LIN {X 0,Y 371.44,Z 415.123,A -85,B 0,C 180,E1 -12712.236,E2 -12712.236} C_VEL
LIN {X 0,Y 371.913,Z 409.005,A -85,B 0,C 180,E1 -12713.675,E2 -12713.675} C_VEL
LIN {X 0,Y 370.1,Z 398.641,A -85,B 0,C 180,E1 -12716.295,E2 -12716.295} C_VEL
LIN {X 0,Y 369.046,Z 393.228,A -85,B 0,C 180,E1 -12717.735,E2 -12717.735} C_VEL
LIN {X 0,Y 368.911,Z 393.034,A -85,B 0,C 180,E1 -12720.987,E2 -12720.987} C_VEL
LIN {X 0,Y 368.937,Z 393.026,A -85,B 0,C 180,E1 -12724.853,E2 -12724.853} C_VEL
LIN {X 0,Y 368.91,Z 393.028,A -85,B 0,C 180,E1 -12728.64,E2 -12728.64} C_VEL
LIN {X 0,Y 368.881,Z 393.034,A -85,B 0,C 180,E1 -12732.009,E2 -12732.009} C_VEL
LIN {X 0,Y 368.953,Z 393.026,A -85,B 0,C 180,E1 -12735.187,E2 -12735.187} C_VEL
LIN {X 0,Y 368.939,Z 393.025,A -85,B 0,C 180,E1 -12738.185,E2 -12738.185} C_VEL
LIN {X 0,Y 368.912,Z 393.034,A -85,B 0,C 180,E1 -12741.358,E2 -12741.358} C_VEL
LIN {X 0,Y 368.934,Z 393.029,A -85,B 0,C 180,E1 -12745.146,E2 -12745.146} C_VEL
LIN {X 0,Y 368.926,Z 393.029,A -85,B 0,C 180,E1 -12749.046,E2 -12749.046} C_VEL
LIN {X 0,Y 368.976,Z 393.025,A -85,B 0,C 180,E1 -12751.563,E2 -12751.563} C_VEL
LIN {X 0,Y 368.996,Z 393.019,A -85,B 0,C 180,E1 -12754.019,E2 -12754.019} C_VEL
LIN {X 0,Y 368.92,Z 393.032,A -85,B 0,C 180,E1 -12757.604,E2 -12757.604} C_VEL
LIN {X 0,Y 368.978,Z 393.024,A -85,B 0,C 180,E1 -12761.107,E2 -12761.107} C_VEL
LIN {X 0,Y 368.993,Z 393.019,A -85,B 0,C 180,E1 -12764.535,E2 -12764.535} C_VEL
LIN {X 0,Y 368.999,Z 393.019,A -85,B 0,C 180,E1 -12767.906,E2 -12767.906} C_VEL
LIN {X 0,Y 369.161,Z 392.999,A -85,B 0,C 180,E1 -12771.869,E2 -12771.869} C_VEL
LIN {X 0,Y 369.138,Z 393.001,A -85,B 0,C 180,E1 -12774.537,E2 -12774.537} C_VEL
LIN {X 0,Y 369.313,Z 392.98,A -85,B 0,C 180,E1 -12777.819,E2 -12777.819} C_VEL
LIN {X 0,Y 369.453,Z 392.962,A -85,B 0,C 180,E1 -12780,E2 -12780} C_VEL
LIN {X 0,Y 369.314,Z 392.978,A -85,B 0,C 180,E1 -12782.181,E2 -12782.181} C_VEL
LIN {X 0,Y 369.192,Z 392.994,A -85,B 0,C 180,E1 -12786.614,E2 -12786.614} C_VEL
LIN {X 0,Y 369.062,Z 393.011,A -85,B 0,C 180,E1 -12789.868,E2 -12789.868} C_VEL
LIN {X 0,Y 369.032,Z 393.015,A -85,B 0,C 180,E1 -12793.772,E2 -12793.772} C_VEL
LIN {X 0,Y 368.996,Z 393.019,A -85,B 0,C 180,E1 -12797.769,E2 -12797.769} C_VEL
LIN {X 0,Y 368.924,Z 393.033,A -85,B 0,C 180,E1 -12801.22,E2 -12801.22} C_VEL
LIN {X 0,Y 368.953,Z 393.026,A -85,B 0,C 180,E1 -12804.776,E2 -12804.776} C_VEL
LIN {X 0,Y 368.983,Z 393.02,A -85,B 0,C 180,E1 -12808.436,E2 -12808.436} C_VEL
LIN {X 0,Y 368.896,Z 393.03,A -85,B 0,C 180,E1 -12812.238,E2 -12812.238} C_VEL
LIN {X 0,Y 368.926,Z 393.032,A -85,B 0,C 180,E1 -12815.002,E2 -12815.002} C_VEL
LIN {X 0,Y 368.907,Z 393.031,A -85,B 0,C 180,E1 -12818.641,E2 -12818.641} C_VEL
LIN {X 0,Y 368.879,Z 393.033,A -85,B 0,C 180,E1 -12822.01,E2 -12822.01} C_VEL
LIN {X 0,Y 368.905,Z 393.035,A -85,B 0,C 180,E1 -12825.18,E2 -12825.18} C_VEL
LIN {X 0,Y 368.908,Z 393.029,A -85,B 0,C 180,E1 -12828.182,E2 -12828.182} C_VEL
LIN {X 0,Y 368.912,Z 393.031,A -85,B 0,C 180,E1 -12831.359,E2 -12831.359} C_VEL
LIN {X 0,Y 368.936,Z 393.031,A -85,B 0,C 180,E1 -12835.147,E2 -12835.147} C_VEL
LIN {X 0,Y 368.929,Z 393.032,A -85,B 0,C 180,E1 -12839.047,E2 -12839.047} C_VEL
LIN {X 0,Y 368.976,Z 393.022,A -85,B 0,C 180,E1 -12841.564,E2 -12841.564} C_VEL
LIN {X 0,Y 369,Z 393.017,A -85,B 0,C 180,E1 -12844.02,E2 -12844.02} C_VEL
LIN {X 0,Y 368.933,Z 393.026,A -85,B 0,C 180,E1 -12847.605,E2 -12847.605} C_VEL
LIN {X 0,Y 368.959,Z 393.027,A -85,B 0,C 180,E1 -12851.106,E2 -12851.106} C_VEL
LIN {X 0,Y 368.999,Z 393.02,A -85,B 0,C 180,E1 -12854.535,E2 -12854.535} C_VEL
LIN {X 0,Y 369.086,Z 393.119,A -85,B 0,C 180,E1 -12857.281,E2 -12857.281} C_VEL
LIN {X 0,Y 371.157,Z 404.31,A -85,B 0,C 180,E1 -12860.381,E2 -12860.381} C_VEL
LIN {X 0,Y 371.305,Z 407.805,A -85,B 0,C 180,E1 -12861.291,E2 -12861.291} C_VEL
LIN {X 0,Y 370.959,Z 411.278,A -85,B 0,C 180,E1 -12862.105,E2 -12862.105} C_VEL
LIN {X 0,Y 371.664,Z 415.551,A -85,B 0,C 180,E1 -12862.281,E2 -12862.281} C_VEL
LIN {X 0,Y 375.657,Z 437.442,A -85,B 0,C 180,E1 -12862.901,E2 -12862.901} C_VEL
LIN {X 0,Y 374.451,Z 518.084,A -85,B 0,C 180,E1 -12864.459,E2 -12864.459} C_VEL
LIN {X 0,Y 373.984,Z 531.756,A -85,B 0,C 180,E1 -12864.943,E2 -12864.943} C_VEL
LIN {X 0,Y 373.319,Z 544.448,A -85,B 0,C 180,E1 -12865.614,E2 -12865.614} C_VEL
LIN {X 0,Y 372.489,Z 556.486,A -85,B 0,C 180,E1 -12866.484,E2 -12866.484} C_VEL
LIN {X 0,Y 371.473,Z 567.981,A -85,B 0,C 180,E1 -12867.56,E2 -12867.56} C_VEL
LIN {X 0,Y 370.657,Z 578.297,A -85,B 0,C 180,E1 -12868.777,E2 -12868.777} C_VEL
LIN {X 0,Y 369.86,Z 586.759,A -85,B 0,C 180,E1 -12870,E2 -12870} C_VEL
LIN {X 0,Y 368.966,Z 595.93,A -85,B 0,C 180,E1 -12871.637,E2 -12871.637} C_VEL
LIN {X 0,Y 368.405,Z 603.301,A -85,B 0,C 180,E1 -12873.281,E2 -12873.281} C_VEL
LIN {X 0,Y 367.91,Z 609.23,A -85,B 0,C 180,E1 -12874.931,E2 -12874.931} C_VEL
LIN {X 0,Y 367.727,Z 613.898,A -85,B 0,C 180,E1 -12876.584,E2 -12876.584} C_VEL
LIN {X 0,Y 367.471,Z 617.474,A -85,B 0,C 180,E1 -12878.246,E2 -12878.246} C_VEL
LIN {X 0,Y 367.268,Z 620.03,A -85,B 0,C 180,E1 -12879.917,E2 -12879.917} C_VEL
LIN {X 0,Y 367.283,Z 621.209,A -85,B 0,C 180,E1 -12881.031,E2 -12881.031} C_VEL
LIN {X 0,Y 367.292,Z 622.145,A -85,B 0,C 180,E1 -12882.613,E2 -12882.613} C_VEL
LIN {X 0,Y 367.18,Z 622.222,A -85,B 0,C 180,E1 -12884.407,E2 -12884.407} C_VEL
LIN {X 0,Y 367.228,Z 621.72,A -85,B 0,C 180,E1 -12885.541,E2 -12885.541} C_VEL
LIN {X 0,Y 367.353,Z 620.477,A -85,B 0,C 180,E1 -12886.973,E2 -12886.973} C_VEL
LIN {X 0,Y 367.665,Z 617.626,A -85,B 0,C 180,E1 -12888.962,E2 -12888.962} C_VEL
LIN {X 0,Y 368.017,Z 614.077,A -85,B 0,C 180,E1 -12890.65,E2 -12890.65} C_VEL
LIN {X 0,Y 368.293,Z 611.729,A -85,B 0,C 180,E1 -12891.537,E2 -12891.537} C_VEL
LIN {X 0,Y 367.938,Z 609.343,A -85,B 0,C 180,E1 -12892.375,E2 -12892.375} C_VEL
LIN {X 0,Y 365.697,Z 605.131,A -85,B 0,C 180,E1 -12893.734,E2 -12893.734} C_VEL
LIN {X 0,Y 363.513,Z 600.325,A -85,B 0,C 180,E1 -12895.054,E2 -12895.054} C_VEL
LIN {X 0,Y 363.247,Z 596.96,A -85,B 0,C 180,E1 -12895.819,E2 -12895.819} C_VEL
LIN {X 0,Y 364.426,Z 588.08,A -85,B 0,C 180,E1 -12897.487,E2 -12897.487} C_VEL
LIN {X 0,Y 365.716,Z 577.768,A -85,B 0,C 180,E1 -12899.027,E2 -12899.027} C_VEL
LIN {X 0,Y 367.063,Z 567.317,A -85,B 0,C 180,E1 -12900.261,E2 -12900.261} C_VEL
LIN {X 0,Y 368.253,Z 555.954,A -85,B 0,C 180,E1 -12901.335,E2 -12901.335} C_VEL
LIN {X 0,Y 369.319,Z 544.043,A -85,B 0,C 180,E1 -12902.196,E2 -12902.196} C_VEL
LIN {X 0,Y 370.206,Z 531.197,A -85,B 0,C 180,E1 -12902.875,E2 -12902.875} C_VEL
LIN {X 0,Y 370.844,Z 517.98,A -85,B 0,C 180,E1 -12903.338,E2 -12903.338} C_VEL
LIN {X 0,Y 372.433,Z 439.897,A -85,B 0,C 180,E1 -12904.888,E2 -12904.888} C_VEL
LIN {X 0,Y 367.754,Z 418.56,A -85,B 0,C 180,E1 -12905.694,E2 -12905.694} C_VEL
LIN {X 0,Y 365.867,Z 412.519,A -85,B 0,C 180,E1 -12905.985,E2 -12905.985} C_VEL
LIN {X 0,Y 365.515,Z 411.249,A -85,B 0,C 180,E1 -12906.142,E2 -12906.142} C_VEL
LIN {X 0,Y 363.427,Z 400.528,A -85,B 0,C 180,E1 -12909.328,E2 -12909.328} C_VEL
LIN {X 0,Y 361.906,Z 393.937,A -85,B 0,C 180,E1 -12911.48,E2 -12911.48} C_VEL
LIN {X 0,Y 361.929,Z 393.903,A -85,B 0,C 180,E1 -12914.35,E2 -12914.35} C_VEL
LIN {X 0,Y 361.882,Z 393.901,A -85,B 0,C 180,E1 -12917.559,E2 -12917.559} C_VEL
LIN {X 0,Y 361.869,Z 393.901,A -85,B 0,C 180,E1 -12920.972,E2 -12920.972} C_VEL
LIN {X 0,Y 361.869,Z 393.9,A -85,B 0,C 180,E1 -12924.654,E2 -12924.654} C_VEL
LIN {X 0,Y 361.853,Z 393.911,A -85,B 0,C 180,E1 -12928.372,E2 -12928.372} C_VEL
LIN {X 0,Y 361.915,Z 393.9,A -85,B 0,C 180,E1 -12932.222,E2 -12932.222} C_VEL
LIN {X 0,Y 361.921,Z 393.9,A -85,B 0,C 180,E1 -12934.709,E2 -12934.709} C_VEL
LIN {X 0,Y 361.894,Z 393.899,A -85,B 0,C 180,E1 -12938.347,E2 -12938.347} C_VEL
LIN {X 0,Y 361.96,Z 393.891,A -85,B 0,C 180,E1 -12942.061,E2 -12942.061} C_VEL
LIN {X 0,Y 361.99,Z 393.886,A -85,B 0,C 180,E1 -12946.101,E2 -12946.101} C_VEL
LIN {X 0,Y 362.028,Z 393.879,A -85,B 0,C 180,E1 -12949.938,E2 -12949.938} C_VEL
LIN {X 0,Y 362.143,Z 393.874,A -85,B 0,C 180,E1 -12952.192,E2 -12952.192} C_VEL
LIN {X 0,Y 362.111,Z 393.87,A -85,B 0,C 180,E1 -12954.431,E2 -12954.431} C_VEL
LIN {X 0,Y 362.282,Z 393.853,A -85,B 0,C 180,E1 -12957.777,E2 -12957.777} C_VEL
LIN {X 0,Y 362.421,Z 393.833,A -85,B 0,C 180,E1 -12960,E2 -12960} C_VEL
LIN {X 0,Y 362.275,Z 393.857,A -85,B 0,C 180,E1 -12962.224,E2 -12962.224} C_VEL
LIN {X 0,Y 362.164,Z 393.875,A -85,B 0,C 180,E1 -12966.686,E2 -12966.686} C_VEL
LIN {X 0,Y 362.067,Z 393.877,A -85,B 0,C 180,E1 -12968.934,E2 -12968.934} C_VEL
LIN {X 0,Y 361.959,Z 393.898,A -85,B 0,C 180,E1 -12972.332,E2 -12972.332} C_VEL
LIN {X 0,Y 361.954,Z 393.892,A -85,B 0,C 180,E1 -12974.621,E2 -12974.621} C_VEL
LIN {X 0,Y 361.952,Z 393.891,A -85,B 0,C 180,E1 -12978.1,E2 -12978.1} C_VEL
LIN {X 0,Y 361.885,Z 393.902,A -85,B 0,C 180,E1 -12981.653,E2 -12981.653} C_VEL
LIN {X 0,Y 361.921,Z 393.9,A -85,B 0,C 180,E1 -12985.291,E2 -12985.291} C_VEL
LIN {X 0,Y 361.912,Z 393.899,A -85,B 0,C 180,E1 -12987.779,E2 -12987.779} C_VEL
LIN {X 0,Y 361.841,Z 393.91,A -85,B 0,C 180,E1 -12991.286,E2 -12991.286} C_VEL
LIN {X 0,Y 361.849,Z 393.907,A -85,B 0,C 180,E1 -12994.281,E2 -12994.281} C_VEL
LIN {X 0,Y 361.861,Z 393.905,A -85,B 0,C 180,E1 -12997.224,E2 -12997.224} C_VEL
LIN {X 0,Y 361.901,Z 393.89,A -85,B 0,C 180,E1 -13000.769,E2 -13000.769} C_VEL
LIN {X 0,Y 361.907,Z 393.907,A -85,B 0,C 180,E1 -13004.355,E2 -13004.355} C_VEL
LIN {X 0,Y 361.837,Z 393.91,A -85,B 0,C 180,E1 -13007.568,E2 -13007.568} C_VEL
LIN {X 0,Y 361.869,Z 393.905,A -85,B 0,C 180,E1 -13010.974,E2 -13010.974} C_VEL
LIN {X 0,Y 361.873,Z 393.91,A -85,B 0,C 180,E1 -13014.656,E2 -13014.656} C_VEL
LIN {X 0,Y 361.836,Z 393.91,A -85,B 0,C 180,E1 -13018.371,E2 -13018.371} C_VEL
LIN {X 0,Y 361.93,Z 394.09,A -85,B 0,C 180,E1 -13019.602,E2 -13019.602} C_VEL
LIN {X 0,Y 364.258,Z 403.929,A -85,B 0,C 180,E1 -13022.564,E2 -13022.564} C_VEL
LIN {X 0,Y 366.125,Z 413.741,A -85,B 0,C 180,E1 -13025.324,E2 -13025.324} C_VEL
LIN {X 0,Y 366.107,Z 417.243,A -85,B 0,C 180,E1 -13026.227,E2 -13026.227} C_VEL
LIN {X 0,Y 365.803,Z 420.538,A -85,B 0,C 180,E1 -13026.993,E2 -13026.993} C_VEL
LIN {X 0,Y 366.882,Z 425.74,A -85,B 0,C 180,E1 -13027.244,E2 -13027.244} C_VEL
LIN {X 0,Y 370.779,Z 444.027,A -85,B 0,C 180,E1 -13027.928,E2 -13027.928} C_VEL
LIN {X 0,Y 372.23,Z 453.66,A -85,B 0,C 180,E1 -13028.238,E2 -13028.238} C_VEL
LIN {X 0,Y 370.734,Z 528.187,A -85,B 0,C 180,E1 -13029.724,E2 -13029.724} C_VEL
LIN {X 0,Y 370.096,Z 541.357,A -85,B 0,C 180,E1 -13030.194,E2 -13030.194} C_VEL
LIN {X 0,Y 369.108,Z 553.473,A -85,B 0,C 180,E1 -13030.826,E2 -13030.826} C_VEL
LIN {X 0,Y 368.082,Z 564.883,A -85,B 0,C 180,E1 -13031.637,E2 -13031.637} C_VEL
LIN {X 0,Y 366.916,Z 575.332,A -85,B 0,C 180,E1 -13032.586,E2 -13032.586} C_VEL
LIN {X 0,Y 365.592,Z 586.073,A -85,B 0,C 180,E1 -13033.816,E2 -13033.816} C_VEL
LIN {X 0,Y 364.426,Z 595.862,A -85,B 0,C 180,E1 -13035.217,E2 -13035.217} C_VEL
LIN {X 0,Y 363.392,Z 603.678,A -85,B 0,C 180,E1 -13036.581,E2 -13036.581} C_VEL
LIN {X 0,Y 362.314,Z 611.495,A -85,B 0,C 180,E1 -13038.249,E2 -13038.249} C_VEL
LIN {X 0,Y 361.558,Z 617.752,A -85,B 0,C 180,E1 -13039.925,E2 -13039.925} C_VEL
LIN {X 0,Y 360.939,Z 622.747,A -85,B 0,C 180,E1 -13041.603,E2 -13041.603} C_VEL
LIN {X 0,Y 360.582,Z 626.625,A -85,B 0,C 180,E1 -13043.285,E2 -13043.285} C_VEL
LIN {X 0,Y 360.381,Z 630.221,A -85,B 0,C 180,E1 -13045.526,E2 -13045.526} C_VEL
LIN {X 0,Y 360.279,Z 631.412,A -85,B 0,C 180,E1 -13046.645,E2 -13046.645} C_VEL
LIN {X 0,Y 360.249,Z 632.531,A -85,B 0,C 180,E1 -13048.882,E2 -13048.882} C_VEL
LIN {X 0,Y 360.29,Z 632.513,A -85,B 0,C 180,E1 -13050,E2 -13050} C_VEL
LIN {X 0,Y 360.251,Z 632.109,A -85,B 0,C 180,E1 -13051.118,E2 -13051.118} C_VEL
LIN {X 0,Y 360.226,Z 631.272,A -85,B 0,C 180,E1 -13052.236,E2 -13052.236} C_VEL
LIN {X 0,Y 360.275,Z 630.026,A -85,B 0,C 180,E1 -13053.355,E2 -13053.355} C_VEL
LIN {X 0,Y 360.353,Z 627.374,A -85,B 0,C 180,E1 -13055.035,E2 -13055.035} C_VEL
LIN {X 0,Y 360.501,Z 623.694,A -85,B 0,C 180,E1 -13056.717,E2 -13056.717} C_VEL
LIN {X 0,Y 360.837,Z 618.886,A -85,B 0,C 180,E1 -13058.4,E2 -13058.4} C_VEL
LIN {X 0,Y 361.294,Z 612.8,A -85,B 0,C 180,E1 -13060.083,E2 -13060.083} C_VEL
LIN {X 0,Y 361.948,Z 605.214,A -85,B 0,C 180,E1 -13061.764,E2 -13061.764} C_VEL
LIN {X 0,Y 362.734,Z 597.46,A -85,B 0,C 180,E1 -13063.159,E2 -13063.159} C_VEL
LIN {X 0,Y 363.644,Z 587.98,A -85,B 0,C 180,E1 -13064.551,E2 -13064.551} C_VEL
LIN {X 0,Y 364.507,Z 577.427,A -85,B 0,C 180,E1 -13065.804,E2 -13065.804} C_VEL
LIN {X 0,Y 365.426,Z 565.676,A -85,B 0,C 180,E1 -13066.911,E2 -13066.911} C_VEL
LIN {X 0,Y 366.366,Z 553.12,A -85,B 0,C 180,E1 -13067.802,E2 -13067.802} C_VEL
LIN {X 0,Y 367.121,Z 539.852,A -85,B 0,C 180,E1 -13068.485,E2 -13068.485} C_VEL
LIN {X 0,Y 367.589,Z 527.842,A -85,B 0,C 180,E1 -13068.895,E2 -13068.895} C_VEL
LIN {X 0,Y 368.647,Z 450.626,A -85,B 0,C 180,E1 -13070.418,E2 -13070.418} C_VEL
LIN {X 0,Y 364.072,Z 420.84,A -85,B 0,C 180,E1 -13071.276,E2 -13071.276} C_VEL
LIN {X 0,Y 364.923,Z 411.05,A -85,B 0,C 180,E1 -13073.554,E2 -13073.554} C_VEL
LIN {X 0,Y 364.068,Z 404.839,A -85,B 0,C 180,E1 -13075.131,E2 -13075.131} C_VEL
LIN {X 0,Y 362.017,Z 394.269,A -85,B 0,C 180,E1 -13077.927,E2 -13077.927} C_VEL
LIN {X 0,Y 361.946,Z 393.899,A -85,B 0,C 180,E1 -13078.248,E2 -13078.248} C_VEL
LIN {X 0,Y 361.838,Z 393.915,A -85,B 0,C 180,E1 -13081.629,E2 -13081.629} C_VEL
LIN {X 0,Y 361.875,Z 393.909,A -85,B 0,C 180,E1 -13085.344,E2 -13085.344} C_VEL
LIN {X 0,Y 361.871,Z 393.907,A -85,B 0,C 180,E1 -13089.026,E2 -13089.026} C_VEL
LIN {X 0,Y 361.838,Z 393.91,A -85,B 0,C 180,E1 -13092.828,E2 -13092.828} C_VEL
LIN {X 0,Y 361.897,Z 393.904,A -85,B 0,C 180,E1 -13095.933,E2 -13095.933} C_VEL
LIN {X 0,Y 361.903,Z 393.905,A -85,B 0,C 180,E1 -13099.231,E2 -13099.231} C_VEL
LIN {X 0,Y 361.867,Z 393.908,A -85,B 0,C 180,E1 -13102.982,E2 -13102.982} C_VEL
LIN {X 0,Y 361.856,Z 393.907,A -85,B 0,C 180,E1 -13106.63,E2 -13106.63} C_VEL
LIN {X 0,Y 361.871,Z 393.909,A -85,B 0,C 180,E1 -13109.672,E2 -13109.672} C_VEL
LIN {X 0,Y 361.951,Z 393.901,A -85,B 0,C 180,E1 -13113.475,E2 -13113.475} C_VEL
LIN {X 0,Y 361.878,Z 393.908,A -85,B 0,C 180,E1 -13117.144,E2 -13117.144} C_VEL
LIN {X 0,Y 361.916,Z 393.9,A -85,B 0,C 180,E1 -13120.724,E2 -13120.724} C_VEL
LIN {X 0,Y 361.941,Z 393.897,A -85,B 0,C 180,E1 -13124.226,E2 -13124.226} C_VEL
LIN {X 0,Y 361.994,Z 393.89,A -85,B 0,C 180,E1 -13126.528,E2 -13126.528} C_VEL
LIN {X 0,Y 362.026,Z 393.887,A -85,B 0,C 180,E1 -13129.938,E2 -13129.938} C_VEL
LIN {X 0,Y 362.157,Z 393.876,A -85,B 0,C 180,E1 -13133.313,E2 -13133.313} C_VEL
LIN {X 0,Y 362.277,Z 393.857,A -85,B 0,C 180,E1 -13137.776,E2 -13137.776} C_VEL
LIN {X 0,Y 362.422,Z 393.837,A -85,B 0,C 180,E1 -13140,E2 -13140} C_VEL
LIN {X 0,Y 362.278,Z 393.855,A -85,B 0,C 180,E1 -13142.223,E2 -13142.223} C_VEL
LIN {X 0,Y 362.159,Z 393.871,A -85,B 0,C 180,E1 -13146.686,E2 -13146.686} C_VEL
LIN {X 0,Y 362.026,Z 393.886,A -85,B 0,C 180,E1 -13150.062,E2 -13150.062} C_VEL
LIN {X 0,Y 361.993,Z 393.891,A -85,B 0,C 180,E1 -13153.899,E2 -13153.899} C_VEL
LIN {X 0,Y 361.963,Z 393.894,A -85,B 0,C 180,E1 -13157.939,E2 -13157.939} C_VEL
LIN {X 0,Y 361.887,Z 393.905,A -85,B 0,C 180,E1 -13161.653,E2 -13161.653} C_VEL
LIN {X 0,Y 361.924,Z 393.904,A -85,B 0,C 180,E1 -13165.29,E2 -13165.29} C_VEL
LIN {X 0,Y 361.919,Z 393.9,A -85,B 0,C 180,E1 -13167.778,E2 -13167.778} C_VEL
LIN {X 0,Y 361.843,Z 393.914,A -85,B 0,C 180,E1 -13171.286,E2 -13171.286} C_VEL
LIN {X 0,Y 361.851,Z 393.908,A -85,B 0,C 180,E1 -13174.281,E2 -13174.281} C_VEL
LIN {X 0,Y 361.862,Z 393.912,A -85,B 0,C 180,E1 -13177.224,E2 -13177.224} C_VEL
LIN {X 0,Y 361.833,Z 393.913,A -85,B 0,C 180,E1 -13180.756,E2 -13180.756} C_VEL
LIN {X 0,Y 361.832,Z 393.911,A -85,B 0,C 180,E1 -13184.366,E2 -13184.366} C_VEL
LIN {X 0,Y 361.854,Z 393.909,A -85,B 0,C 180,E1 -13187.565,E2 -13187.565} C_VEL
LIN {X 0,Y 361.874,Z 393.911,A -85,B 0,C 180,E1 -13190.973,E2 -13190.973} C_VEL
LIN {X 0,Y 361.874,Z 393.908,A -85,B 0,C 180,E1 -13194.655,E2 -13194.655} C_VEL
LIN {X 0,Y 361.837,Z 393.91,A -85,B 0,C 180,E1 -13198.371,E2 -13198.371} C_VEL
LIN {X 0,Y 361.9,Z 393.908,A -85,B 0,C 180,E1 -13200.956,E2 -13200.956} C_VEL
LIN {X 0,Y 361.954,Z 393.897,A -85,B 0,C 180,E1 -13203.475,E2 -13203.475} C_VEL
LIN {X 0,Y 361.891,Z 393.907,A -85,B 0,C 180,E1 -13207.145,E2 -13207.145} C_VEL
LIN {X 0,Y 361.908,Z 393.905,A -85,B 0,C 180,E1 -13210.724,E2 -13210.724} C_VEL
LIN {X 0,Y 361.934,Z 393.902,A -85,B 0,C 180,E1 -13213.066,E2 -13213.066} C_VEL
LIN {X 0,Y 362.053,Z 393.976,A -85,B 0,C 180,E1 -13217.03,E2 -13217.03} C_VEL
LIN {X 0,Y 364.341,Z 406.519,A -85,B 0,C 180,E1 -13220.563,E2 -13220.563} C_VEL
LIN {X 0,Y 364.143,Z 411.267,A -85,B 0,C 180,E1 -13221.747,E2 -13221.747} C_VEL
LIN {X 0,Y 364.313,Z 413.493,A -85,B 0,C 180,E1 -13221.875,E2 -13221.875} C_VEL
LIN {X 0,Y 368.927,Z 439.229,A -85,B 0,C 180,E1 -13222.618,E2 -13222.618} C_VEL
LIN {X 0,Y 367.614,Z 518.872,A -85,B 0,C 180,E1 -13224.188,E2 -13224.188} C_VEL
LIN {X 0,Y 367.077,Z 532.529,A -85,B 0,C 180,E1 -13224.689,E2 -13224.689} C_VEL
LIN {X 0,Y 366.387,Z 545.345,A -85,B 0,C 180,E1 -13225.392,E2 -13225.392} C_VEL
LIN {X 0,Y 365.544,Z 557.165,A -85,B 0,C 180,E1 -13226.279,E2 -13226.279} C_VEL
LIN {X 0,Y 364.495,Z 568.557,A -85,B 0,C 180,E1 -13227.375,E2 -13227.375} C_VEL
LIN {X 0,Y 363.656,Z 578.783,A -85,B 0,C 180,E1 -13228.615,E2 -13228.615} C_VEL
LIN {X 0,Y 362.751,Z 587.996,A -85,B 0,C 180,E1 -13230,E2 -13230} C_VEL
LIN {X 0,Y 361.864,Z 596.958,A -85,B 0,C 180,E1 -13231.669,E2 -13231.669} C_VEL
LIN {X 0,Y 361.29,Z 604.167,A -85,B 0,C 180,E1 -13233.345,E2 -13233.345} C_VEL
LIN {X 0,Y 360.824,Z 609.932,A -85,B 0,C 180,E1 -13235.028,E2 -13235.028} C_VEL
LIN {X 0,Y 360.596,Z 614.466,A -85,B 0,C 180,E1 -13236.715,E2 -13236.715} C_VEL
LIN {X 0,Y 360.438,Z 616.864,A -85,B 0,C 180,E1 -13237.844,E2 -13237.844} C_VEL
LIN {X 0,Y 360.268,Z 618.833,A -85,B 0,C 180,E1 -13238.978,E2 -13238.978} C_VEL
LIN {X 0,Y 360.163,Z 620.376,A -85,B 0,C 180,E1 -13240.114,E2 -13240.114} C_VEL
LIN {X 0,Y 360.177,Z 621.451,A -85,B 0,C 180,E1 -13241.252,E2 -13241.252} C_VEL
LIN {X 0,Y 360.205,Z 622.257,A -85,B 0,C 180,E1 -13242.695,E2 -13242.695} C_VEL
LIN {X 0,Y 360.095,Z 622.269,A -85,B 0,C 180,E1 -13244.697,E2 -13244.697} C_VEL
LIN {X 0,Y 360.167,Z 621.68,A -85,B 0,C 180,E1 -13245.853,E2 -13245.853} C_VEL
LIN {X 0,Y 360.297,Z 620.6,A -85,B 0,C 180,E1 -13247.098,E2 -13247.098} C_VEL
LIN {X 0,Y 360.45,Z 619.268,A -85,B 0,C 180,E1 -13248.177,E2 -13248.177} C_VEL
LIN {X 0,Y 360.768,Z 616.239,A -85,B 0,C 180,E1 -13249.932,E2 -13249.932} C_VEL
LIN {X 0,Y 361.261,Z 612.074,A -85,B 0,C 180,E1 -13251.692,E2 -13251.692} C_VEL
LIN {X 0,Y 362.046,Z 605.568,A -85,B 0,C 180,E1 -13253.752,E2 -13253.752} C_VEL
LIN {X 0,Y 363.006,Z 598.411,A -85,B 0,C 180,E1 -13255.516,E2 -13255.516} C_VEL
LIN {X 0,Y 363.247,Z 596.96,A -85,B 0,C 180,E1 -13255.819,E2 -13255.819} C_VEL
LIN {X 0,Y 362.999,Z 593.432,A -85,B 0,C 180,E1 -13256.567,E2 -13256.567} C_VEL
LIN {X 0,Y 360.979,Z 587.458,A -85,B 0,C 180,E1 -13257.786,E2 -13257.786} C_VEL
LIN {X 0,Y 359.151,Z 580.987,A -85,B 0,C 180,E1 -13258.94,E2 -13258.94} C_VEL
LIN {X 0,Y 359.183,Z 576.611,A -85,B 0,C 180,E1 -13259.572,E2 -13259.572} C_VEL
LIN {X 0,Y 360.606,Z 565.776,A -85,B 0,C 180,E1 -13260.84,E2 -13260.84} C_VEL
LIN {X 0,Y 361.725,Z 555.469,A -85,B 0,C 180,E1 -13261.803,E2 -13261.803} C_VEL
LIN {X 0,Y 362.819,Z 543.335,A -85,B 0,C 180,E1 -13262.679,E2 -13262.679} C_VEL
LIN {X 0,Y 363.766,Z 530.221,A -85,B 0,C 180,E1 -13263.367,E2 -13263.367} C_VEL
LIN {X 0,Y 364.398,Z 517.585,A -85,B 0,C 180,E1 -13263.799,E2 -13263.799} C_VEL
LIN {X 0,Y 365.977,Z 440.622,A -85,B 0,C 180,E1 -13265.354,E2 -13265.354} C_VEL
LIN {X 0,Y 361.106,Z 418.719,A -85,B 0,C 180,E1 -13266.218,E2 -13266.218} C_VEL
LIN {X 0,Y 358.451,Z 411.884,A -85,B 0,C 180,E1 -13266.627,E2 -13266.627} C_VEL
LIN {X 0,Y 357.191,Z 405.438,A -85,B 0,C 180,E1 -13268.506,E2 -13268.506} C_VEL
LIN {X 0,Y 355.277,Z 396.751,A -85,B 0,C 180,E1 -13271.262,E2 -13271.262} C_VEL
LIN {X 0,Y 354.868,Z 394.807,A -85,B 0,C 180,E1 -13271.983,E2 -13271.983} C_VEL
LIN {X 0,Y 354.883,Z 394.775,A -85,B 0,C 180,E1 -13275.473,E2 -13275.473} C_VEL
LIN {X 0,Y 354.851,Z 394.783,A -85,B 0,C 180,E1 -13279.188,E2 -13279.188} C_VEL
LIN {X 0,Y 354.804,Z 394.786,A -85,B 0,C 180,E1 -13282.401,E2 -13282.401} C_VEL
LIN {X 0,Y 354.806,Z 394.777,A -85,B 0,C 180,E1 -13284.94,E2 -13284.94} C_VEL
LIN {X 0,Y 354.809,Z 394.789,A -85,B 0,C 180,E1 -13288.399,E2 -13288.399} C_VEL
LIN {X 0,Y 354.847,Z 394.777,A -85,B 0,C 180,E1 -13291.619,E2 -13291.619} C_VEL
LIN {X 0,Y 354.892,Z 394.776,A -85,B 0,C 180,E1 -13294.172,E2 -13294.172} C_VEL
LIN {X 0,Y 354.834,Z 394.778,A -85,B 0,C 180,E1 -13297.894,E2 -13297.894} C_VEL
LIN {X 0,Y 354.916,Z 394.768,A -85,B 0,C 180,E1 -13301.891,E2 -13301.891} C_VEL
LIN {X 0,Y 354.935,Z 394.765,A -85,B 0,C 180,E1 -13305.981,E2 -13305.981} C_VEL
LIN {X 0,Y 354.975,Z 394.757,A -85,B 0,C 180,E1 -13309.736,E2 -13309.736} C_VEL
LIN {X 0,Y 355.106,Z 394.75,A -85,B 0,C 180,E1 -13312.037,E2 -13312.037} C_VEL
LIN {X 0,Y 355.086,Z 394.745,A -85,B 0,C 180,E1 -13314.321,E2 -13314.321} C_VEL
LIN {X 0,Y 355.246,Z 394.73,A -85,B 0,C 180,E1 -13317.732,E2 -13317.732} C_VEL
LIN {X 0,Y 355.391,Z 394.709,A -85,B 0,C 180,E1 -13320,E2 -13320} C_VEL
LIN {X 0,Y 355.238,Z 394.734,A -85,B 0,C 180,E1 -13322.268,E2 -13322.268} C_VEL
LIN {X 0,Y 355.13,Z 394.749,A -85,B 0,C 180,E1 -13326.819,E2 -13326.819} C_VEL
LIN {X 0,Y 355.009,Z 394.756,A -85,B 0,C 180,E1 -13329.113,E2 -13329.113} C_VEL
LIN {X 0,Y 354.919,Z 394.771,A -85,B 0,C 180,E1 -13332.581,E2 -13332.581} C_VEL
LIN {X 0,Y 354.882,Z 394.778,A -85,B 0,C 180,E1 -13336.096,E2 -13336.096} C_VEL
LIN {X 0,Y 354.899,Z 394.769,A -85,B 0,C 180,E1 -13338.472,E2 -13338.472} C_VEL
LIN {X 0,Y 354.828,Z 394.782,A -85,B 0,C 180,E1 -13342.107,E2 -13342.107} C_VEL
LIN {X 0,Y 354.892,Z 394.775,A -85,B 0,C 180,E1 -13345.828,E2 -13345.828} C_VEL
LIN {X 0,Y 354.848,Z 394.78,A -85,B 0,C 180,E1 -13349.679,E2 -13349.679} C_VEL
LIN {X 0,Y 354.801,Z 394.785,A -85,B 0,C 180,E1 -13353.703,E2 -13353.703} C_VEL
LIN {X 0,Y 354.794,Z 394.79,A -85,B 0,C 180,E1 -13356.46,E2 -13356.46} C_VEL
LIN {X 0,Y 354.819,Z 394.785,A -85,B 0,C 180,E1 -13359.425,E2 -13359.425} C_VEL
LIN {X 0,Y 354.831,Z 394.777,A -85,B 0,C 180,E1 -13362.876,E2 -13362.876} C_VEL
LIN {X 0,Y 354.78,Z 394.78,A -85,B 0,C 180,E1 -13366.107,E2 -13366.107} C_VEL
LIN {X 0,Y 354.804,Z 394.785,A -85,B 0,C 180,E1 -13369.183,E2 -13369.183} C_VEL
LIN {X 0,Y 354.806,Z 394.788,A -85,B 0,C 180,E1 -13372.403,E2 -13372.403} C_VEL
LIN {X 0,Y 354.81,Z 394.789,A -85,B 0,C 180,E1 -13374.942,E2 -13374.942} C_VEL
LIN {X 0,Y 354.885,Z 394.969,A -85,B 0,C 180,E1 -13379.102,E2 -13379.102} C_VEL
LIN {X 0,Y 357.495,Z 405.982,A -85,B 0,C 180,E1 -13382.494,E2 -13382.494} C_VEL
LIN {X 0,Y 359.38,Z 416.303,A -85,B 0,C 180,E1 -13385.446,E2 -13385.446} C_VEL
LIN {X 0,Y 359.114,Z 420.596,A -85,B 0,C 180,E1 -13386.472,E2 -13386.472} C_VEL
LIN {X 0,Y 363.088,Z 438.438,A -85,B 0,C 180,E1 -13387.225,E2 -13387.225} C_VEL
LIN {X 0,Y 365.818,Z 454.238,A -85,B 0,C 180,E1 -13387.777,E2 -13387.777} C_VEL
LIN {X 0,Y 364.251,Z 528.074,A -85,B 0,C 180,E1 -13389.273,E2 -13389.273} C_VEL
LIN {X 0,Y 363.587,Z 541.247,A -85,B 0,C 180,E1 -13389.751,E2 -13389.751} C_VEL
LIN {X 0,Y 362.572,Z 553.364,A -85,B 0,C 180,E1 -13390.393,E2 -13390.393} C_VEL
LIN {X 0,Y 361.401,Z 565.606,A -85,B 0,C 180,E1 -13391.285,E2 -13391.285} C_VEL
LIN {X 0,Y 360.013,Z 577.156,A -85,B 0,C 180,E1 -13392.388,E2 -13392.388} C_VEL
LIN {X 0,Y 358.658,Z 587.564,A -85,B 0,C 180,E1 -13393.641,E2 -13393.641} C_VEL
LIN {X 0,Y 357.376,Z 597.766,A -85,B 0,C 180,E1 -13395.188,E2 -13395.188} C_VEL
LIN {X 0,Y 356.271,Z 605.34,A -85,B 0,C 180,E1 -13396.598,E2 -13396.598} C_VEL
LIN {X 0,Y 355.21,Z 612.777,A -85,B 0,C 180,E1 -13398.3,E2 -13398.3} C_VEL
LIN {X 0,Y 354.331,Z 619.667,A -85,B 0,C 180,E1 -13400.294,E2 -13400.294} C_VEL
LIN {X 0,Y 353.74,Z 624.23,A -85,B 0,C 180,E1 -13402.006,E2 -13402.006} C_VEL
LIN {X 0,Y 353.389,Z 628.047,A -85,B 0,C 180,E1 -13403.921,E2 -13403.921} C_VEL
LIN {X 0,Y 353.297,Z 630.203,A -85,B 0,C 180,E1 -13405.436,E2 -13405.436} C_VEL
LIN {X 0,Y 353.204,Z 631.364,A -85,B 0,C 180,E1 -13406.578,E2 -13406.578} C_VEL
LIN {X 0,Y 353.149,Z 632.439,A -85,B 0,C 180,E1 -13408.86,E2 -13408.86} C_VEL
LIN {X 0,Y 353.191,Z 632.403,A -85,B 0,C 180,E1 -13410,E2 -13410} C_VEL
LIN {X 0,Y 353.15,Z 631.973,A -85,B 0,C 180,E1 -13411.141,E2 -13411.141} C_VEL
LIN {X 0,Y 353.199,Z 629.842,A -85,B 0,C 180,E1 -13413.422,E2 -13413.422} C_VEL
LIN {X 0,Y 353.258,Z 627.15,A -85,B 0,C 180,E1 -13415.137,E2 -13415.137} C_VEL
LIN {X 0,Y 353.421,Z 623.427,A -85,B 0,C 180,E1 -13416.853,E2 -13416.853} C_VEL
LIN {X 0,Y 353.793,Z 618.575,A -85,B 0,C 180,E1 -13418.568,E2 -13418.568} C_VEL
LIN {X 0,Y 354.278,Z 612.439,A -85,B 0,C 180,E1 -13420.285,E2 -13420.285} C_VEL
LIN {X 0,Y 354.964,Z 604.796,A -85,B 0,C 180,E1 -13421.999,E2 -13421.999} C_VEL
LIN {X 0,Y 355.769,Z 596.965,A -85,B 0,C 180,E1 -13423.422,E2 -13423.422} C_VEL
LIN {X 0,Y 356.706,Z 587.377,A -85,B 0,C 180,E1 -13424.841,E2 -13424.841} C_VEL
LIN {X 0,Y 357.631,Z 576.714,A -85,B 0,C 180,E1 -13426.116,E2 -13426.116} C_VEL
LIN {X 0,Y 358.456,Z 566.417,A -85,B 0,C 180,E1 -13427.103,E2 -13427.103} C_VEL
LIN {X 0,Y 359.427,Z 554.21,A -85,B 0,C 180,E1 -13428.01,E2 -13428.01} C_VEL
LIN {X 0,Y 360.245,Z 540.581,A -85,B 0,C 180,E1 -13428.741,E2 -13428.741} C_VEL
LIN {X 0,Y 360.763,Z 527.84,A -85,B 0,C 180,E1 -13429.192,E2 -13429.192} C_VEL
LIN {X 0,Y 361.852,Z 451.493,A -85,B 0,C 180,E1 -13430.726,E2 -13430.726} C_VEL
LIN {X 0,Y 357.186,Z 420.833,A -85,B 0,C 180,E1 -13431.619,E2 -13431.619} C_VEL
LIN {X 0,Y 357.543,Z 415.982,A -85,B 0,C 180,E1 -13432.726,E2 -13432.726} C_VEL
LIN {X 0,Y 357.864,Z 410.622,A -85,B 0,C 180,E1 -13434.048,E2 -13434.048} C_VEL
LIN {X 0,Y 355.68,Z 398.608,A -85,B 0,C 180,E1 -13437.23,E2 -13437.23} C_VEL
LIN {X 0,Y 354.928,Z 394.826,A -85,B 0,C 180,E1 -13438.335,E2 -13438.335} C_VEL
LIN {X 0,Y 354.787,Z 394.788,A -85,B 0,C 180,E1 -13442.333,E2 -13442.333} C_VEL
LIN {X 0,Y 354.822,Z 394.788,A -85,B 0,C 180,E1 -13445.699,E2 -13445.699} C_VEL
LIN {X 0,Y 354.824,Z 394.788,A -85,B 0,C 180,E1 -13449.423,E2 -13449.423} C_VEL
LIN {X 0,Y 354.79,Z 394.788,A -85,B 0,C 180,E1 -13452.867,E2 -13452.867} C_VEL
LIN {X 0,Y 354.839,Z 394.781,A -85,B 0,C 180,E1 -13456.115,E2 -13456.115} C_VEL
LIN {X 0,Y 354.854,Z 394.782,A -85,B 0,C 180,E1 -13459.188,E2 -13459.188} C_VEL
LIN {X 0,Y 354.807,Z 394.785,A -85,B 0,C 180,E1 -13462.402,E2 -13462.402} C_VEL
LIN {X 0,Y 354.81,Z 394.786,A -85,B 0,C 180,E1 -13464.94,E2 -13464.94} C_VEL
LIN {X 0,Y 354.79,Z 394.787,A -85,B 0,C 180,E1 -13468.405,E2 -13468.405} C_VEL
LIN {X 0,Y 354.848,Z 394.784,A -85,B 0,C 180,E1 -13471.619,E2 -13471.619} C_VEL
LIN {X 0,Y 354.895,Z 394.774,A -85,B 0,C 180,E1 -13474.172,E2 -13474.172} C_VEL
LIN {X 0,Y 354.813,Z 394.786,A -85,B 0,C 180,E1 -13477.892,E2 -13477.892} C_VEL
LIN {X 0,Y 354.919,Z 394.773,A -85,B 0,C 180,E1 -13481.891,E2 -13481.891} C_VEL
LIN {X 0,Y 354.938,Z 394.77,A -85,B 0,C 180,E1 -13485.981,E2 -13485.981} C_VEL
LIN {X 0,Y 354.973,Z 394.766,A -85,B 0,C 180,E1 -13489.736,E2 -13489.736} C_VEL
LIN {X 0,Y 355.121,Z 394.751,A -85,B 0,C 180,E1 -13493.18,E2 -13493.18} C_VEL
LIN {X 0,Y 355.241,Z 394.733,A -85,B 0,C 180,E1 -13497.732,E2 -13497.732} C_VEL
LIN {X 0,Y 355.392,Z 394.712,A -85,B 0,C 180,E1 -13500,E2 -13500} C_VEL
LIN {X 0,Y 355.241,Z 394.731,A -85,B 0,C 180,E1 -13502.268,E2 -13502.268} C_VEL
LIN {X 0,Y 355.122,Z 394.748,A -85,B 0,C 180,E1 -13506.819,E2 -13506.819} C_VEL
LIN {X 0,Y 354.973,Z 394.764,A -85,B 0,C 180,E1 -13510.264,E2 -13510.264} C_VEL
LIN {X 0,Y 354.938,Z 394.769,A -85,B 0,C 180,E1 -13514.019,E2 -13514.019} C_VEL
LIN {X 0,Y 354.918,Z 394.771,A -85,B 0,C 180,E1 -13518.108,E2 -13518.108} C_VEL
LIN {X 0,Y 354.83,Z 394.782,A -85,B 0,C 180,E1 -13522.106,E2 -13522.106} C_VEL
LIN {X 0,Y 354.895,Z 394.775,A -85,B 0,C 180,E1 -13525.828,E2 -13525.828} C_VEL
LIN {X 0,Y 354.851,Z 394.781,A -85,B 0,C 180,E1 -13529.679,E2 -13529.679} C_VEL
LIN {X 0,Y 354.803,Z 394.786,A -85,B 0,C 180,E1 -13533.702,E2 -13533.702} C_VEL
LIN {X 0,Y 354.795,Z 394.787,A -85,B 0,C 180,E1 -13536.46,E2 -13536.46} C_VEL
LIN {X 0,Y 354.821,Z 394.786,A -85,B 0,C 180,E1 -13539.424,E2 -13539.424} C_VEL
LIN {X 0,Y 354.786,Z 394.791,A -85,B 0,C 180,E1 -13542.868,E2 -13542.868} C_VEL
LIN {X 0,Y 354.781,Z 394.788,A -85,B 0,C 180,E1 -13546.107,E2 -13546.107} C_VEL
LIN {X 0,Y 354.823,Z 394.788,A -85,B 0,C 180,E1 -13549.185,E2 -13549.185} C_VEL
LIN {X 0,Y 354.808,Z 394.786,A -85,B 0,C 180,E1 -13552.402,E2 -13552.402} C_VEL
LIN {X 0,Y 354.812,Z 394.79,A -85,B 0,C 180,E1 -13554.941,E2 -13554.941} C_VEL
LIN {X 0,Y 354.792,Z 394.787,A -85,B 0,C 180,E1 -13558.406,E2 -13558.406} C_VEL
LIN {X 0,Y 354.849,Z 394.781,A -85,B 0,C 180,E1 -13561.619,E2 -13561.619} C_VEL
LIN {X 0,Y 354.899,Z 394.774,A -85,B 0,C 180,E1 -13564.173,E2 -13564.173} C_VEL
LIN {X 0,Y 354.835,Z 394.782,A -85,B 0,C 180,E1 -13567.894,E2 -13567.894} C_VEL
LIN {X 0,Y 354.923,Z 394.77,A -85,B 0,C 180,E1 -13571.892,E2 -13571.892} C_VEL
LIN {X 0,Y 354.944,Z 394.771,A -85,B 0,C 180,E1 -13575.981,E2 -13575.981} C_VEL
LIN {X 0,Y 355.021,Z 394.965,A -85,B 0,C 180,E1 -13576.841,E2 -13576.841} C_VEL
LIN {X 0,Y 357.332,Z 407.505,A -85,B 0,C 180,E1 -13580.414,E2 -13580.414} C_VEL
LIN {X 0,Y 357.297,Z 411.431,A -85,B 0,C 180,E1 -13581.41,E2 -13581.41} C_VEL
LIN {X 0,Y 357.804,Z 415.872,A -85,B 0,C 180,E1 -13581.587,E2 -13581.587} C_VEL
LIN {X 0,Y 362.128,Z 439.956,A -85,B 0,C 180,E1 -13582.303,E2 -13582.303} C_VEL
LIN {X 0,Y 360.773,Z 519.01,A -85,B 0,C 180,E1 -13583.89,E2 -13583.89} C_VEL
LIN {X 0,Y 360.304,Z 531.824,A -85,B 0,C 180,E1 -13584.364,E2 -13584.364} C_VEL
LIN {X 0,Y 359.549,Z 545.118,A -85,B 0,C 180,E1 -13585.094,E2 -13585.094} C_VEL
LIN {X 0,Y 358.739,Z 556.239,A -85,B 0,C 180,E1 -13585.927,E2 -13585.927} C_VEL
LIN {X 0,Y 357.659,Z 567.82,A -85,B 0,C 180,E1 -13587.043,E2 -13587.043} C_VEL
LIN {X 0,Y 356.719,Z 578.216,A -85,B 0,C 180,E1 -13588.306,E2 -13588.306} C_VEL
LIN {X 0,Y 355.803,Z 587.58,A -85,B 0,C 180,E1 -13589.717,E2 -13589.717} C_VEL
LIN {X 0,Y 354.873,Z 596.63,A -85,B 0,C 180,E1 -13591.418,E2 -13591.418} C_VEL
LIN {X 0,Y 354.262,Z 603.916,A -85,B 0,C 180,E1 -13593.127,E2 -13593.127} C_VEL
LIN {X 0,Y 353.775,Z 608.861,A -85,B 0,C 180,E1 -13594.557,E2 -13594.557} C_VEL
LIN {X 0,Y 353.572,Z 613.842,A -85,B 0,C 180,E1 -13596.354,E2 -13596.354} C_VEL
LIN {X 0,Y 353.316,Z 617.334,A -85,B 0,C 180,E1 -13598.003,E2 -13598.003} C_VEL
LIN {X 0,Y 353.154,Z 619.244,A -85,B 0,C 180,E1 -13599.16,E2 -13599.16} C_VEL
LIN {X 0,Y 353.066,Z 620.677,A -85,B 0,C 180,E1 -13600.32,E2 -13600.32} C_VEL
LIN {X 0,Y 353.071,Z 621.692,A -85,B 0,C 180,E1 -13601.481,E2 -13601.481} C_VEL
LIN {X 0,Y 353.116,Z 622.368,A -85,B 0,C 180,E1 -13602.777,E2 -13602.777} C_VEL
LIN {X 0,Y 353.003,Z 622.286,A -85,B 0,C 180,E1 -13604.999,E2 -13604.999} C_VEL
LIN {X 0,Y 353.214,Z 620.707,A -85,B 0,C 180,E1 -13607.24,E2 -13607.24} C_VEL
LIN {X 0,Y 353.405,Z 619.06,A -85,B 0,C 180,E1 -13608.552,E2 -13608.552} C_VEL
LIN {X 0,Y 353.782,Z 615.907,A -85,B 0,C 180,E1 -13610.343,E2 -13610.343} C_VEL
LIN {X 0,Y 354.325,Z 611.602,A -85,B 0,C 180,E1 -13612.139,E2 -13612.139} C_VEL
LIN {X 0,Y 355.073,Z 606.008,A -85,B 0,C 180,E1 -13613.938,E2 -13613.938} C_VEL
LIN {X 0,Y 356.075,Z 598.933,A -85,B 0,C 180,E1 -13615.735,E2 -13615.735} C_VEL
LIN {X 0,Y 357.291,Z 590.638,A -85,B 0,C 180,E1 -13617.411,E2 -13617.411} C_VEL
LIN {X 0,Y 358.63,Z 580.69,A -85,B 0,C 180,E1 -13619.013,E2 -13619.013} C_VEL
LIN {X 0,Y 359.183,Z 576.611,A -85,B 0,C 180,E1 -13619.572,E2 -13619.572} C_VEL
LIN {X 0,Y 358.982,Z 573.63,A -85,B 0,C 180,E1 -13619.994,E2 -13619.994} C_VEL
LIN {X 0,Y 356.872,Z 569.015,A -85,B 0,C 180,E1 -13620.714,E2 -13620.714} C_VEL
LIN {X 0,Y 354.755,Z 564.211,A -85,B 0,C 180,E1 -13621.4,E2 -13621.4} C_VEL
LIN {X 0,Y 354.526,Z 560.916,A -85,B 0,C 180,E1 -13621.76,E2 -13621.76} C_VEL
LIN {X 0,Y 355.766,Z 549.245,A -85,B 0,C 180,E1 -13622.736,E2 -13622.736} C_VEL
LIN {X 0,Y 356.867,Z 536.399,A -85,B 0,C 180,E1 -13623.538,E2 -13623.538} C_VEL
LIN {X 0,Y 357.704,Z 523.844,A -85,B 0,C 180,E1 -13624.081,E2 -13624.081} C_VEL
LIN {X 0,Y 358.209,Z 509.211,A -85,B 0,C 180,E1 -13624.454,E2 -13624.454} C_VEL
LIN {X 0,Y 359.558,Z 441.592,A -85,B 0,C 180,E1 -13625.837,E2 -13625.837} C_VEL
LIN {X 0,Y 355.087,Z 421.314,A -85,B 0,C 180,E1 -13626.659,E2 -13626.659} C_VEL
LIN {X 0,Y 351.333,Z 412.068,A -85,B 0,C 180,E1 -13627.225,E2 -13627.225} C_VEL
LIN {X 0,Y 350.43,Z 407.526,A -85,B 0,C 180,E1 -13628.541,E2 -13628.541} C_VEL
LIN {X 0,Y 348.265,Z 397.626,A -85,B 0,C 180,E1 -13631.753,E2 -13631.753} C_VEL
LIN {X 0,Y 347.795,Z 395.683,A -85,B 0,C 180,E1 -13632.503,E2 -13632.503} C_VEL
LIN {X 0,Y 347.826,Z 395.654,A -85,B 0,C 180,E1 -13635.005,E2 -13635.005} C_VEL
LIN {X 0,Y 347.78,Z 395.656,A -85,B 0,C 180,E1 -13638.39,E2 -13638.39} C_VEL
LIN {X 0,Y 347.771,Z 395.659,A -85,B 0,C 180,E1 -13642.01,E2 -13642.01} C_VEL
LIN {X 0,Y 347.738,Z 395.656,A -85,B 0,C 180,E1 -13645.535,E2 -13645.535} C_VEL
LIN {X 0,Y 347.758,Z 395.667,A -85,B 0,C 180,E1 -13648.302,E2 -13648.302} C_VEL
LIN {X 0,Y 347.799,Z 395.646,A -85,B 0,C 180,E1 -13650.99,E2 -13650.99} C_VEL
LIN {X 0,Y 347.825,Z 395.657,A -85,B 0,C 180,E1 -13653.607,E2 -13653.607} C_VEL
LIN {X 0,Y 347.783,Z 395.663,A -85,B 0,C 180,E1 -13656.162,E2 -13656.162} C_VEL
LIN {X 0,Y 347.824,Z 395.657,A -85,B 0,C 180,E1 -13659.91,E2 -13659.91} C_VEL
LIN {X 0,Y 347.859,Z 395.648,A -85,B 0,C 180,E1 -13662.359,E2 -13662.359} C_VEL
LIN {X 0,Y 347.89,Z 395.643,A -85,B 0,C 180,E1 -13665.971,E2 -13665.971} C_VEL
LIN {X 0,Y 347.925,Z 395.636,A -85,B 0,C 180,E1 -13669.526,E2 -13669.526} C_VEL
LIN {X 0,Y 348.066,Z 395.627,A -85,B 0,C 180,E1 -13671.875,E2 -13671.875} C_VEL
LIN {X 0,Y 348.061,Z 395.62,A -85,B 0,C 180,E1 -13674.206,E2 -13674.206} C_VEL
LIN {X 0,Y 348.209,Z 395.606,A -85,B 0,C 180,E1 -13677.687,E2 -13677.687} C_VEL
LIN {X 0,Y 348.36,Z 395.585,A -85,B 0,C 180,E1 -13680,E2 -13680} C_VEL
LIN {X 0,Y 348.201,Z 395.611,A -85,B 0,C 180,E1 -13682.314,E2 -13682.314} C_VEL
LIN {X 0,Y 348.098,Z 395.623,A -85,B 0,C 180,E1 -13686.958,E2 -13686.958} C_VEL
LIN {X 0,Y 347.961,Z 395.634,A -85,B 0,C 180,E1 -13689.299,E2 -13689.299} C_VEL
LIN {X 0,Y 347.886,Z 395.643,A -85,B 0,C 180,E1 -13692.84,E2 -13692.84} C_VEL
LIN {X 0,Y 347.832,Z 395.659,A -85,B 0,C 180,E1 -13696.432,E2 -13696.432} C_VEL
LIN {X 0,Y 347.849,Z 395.649,A -85,B 0,C 180,E1 -13698.861,E2 -13698.861} C_VEL
LIN {X 0,Y 347.768,Z 395.658,A -85,B 0,C 180,E1 -13702.58,E2 -13702.58} C_VEL
LIN {X 0,Y 347.805,Z 395.659,A -85,B 0,C 180,E1 -13705.109,E2 -13705.109} C_VEL
LIN {X 0,Y 347.804,Z 395.656,A -85,B 0,C 180,E1 -13707.695,E2 -13707.695} C_VEL
LIN {X 0,Y 347.758,Z 395.662,A -85,B 0,C 180,E1 -13710.347,E2 -13710.347} C_VEL
LIN {X 0,Y 347.739,Z 395.665,A -85,B 0,C 180,E1 -13714.465,E2 -13714.465} C_VEL
LIN {X 0,Y 347.772,Z 395.661,A -85,B 0,C 180,E1 -13717.99,E2 -13717.99} C_VEL
LIN {X 0,Y 347.78,Z 395.644,A -85,B 0,C 180,E1 -13721.61,E2 -13721.61} C_VEL
LIN {X 0,Y 347.793,Z 395.657,A -85,B 0,C 180,E1 -13725.013,E2 -13725.013} C_VEL
LIN {X 0,Y 347.754,Z 395.67,A -85,B 0,C 180,E1 -13728.397,E2 -13728.397} C_VEL
LIN {X 0,Y 347.772,Z 395.667,A -85,B 0,C 180,E1 -13732.012,E2 -13732.012} C_VEL
LIN {X 0,Y 347.743,Z 395.666,A -85,B 0,C 180,E1 -13735.537,E2 -13735.537} C_VEL
LIN {X 0,Y 347.753,Z 395.706,A -85,B 0,C 180,E1 -13738.472,E2 -13738.472} C_VEL
LIN {X 0,Y 348.865,Z 400.3,A -85,B 0,C 180,E1 -13740.026,E2 -13740.026} C_VEL
LIN {X 0,Y 351.054,Z 409.671,A -85,B 0,C 180,E1 -13742.907,E2 -13742.907} C_VEL
LIN {X 0,Y 352.493,Z 417.724,A -85,B 0,C 180,E1 -13745.249,E2 -13745.249} C_VEL
LIN {X 0,Y 352.422,Z 420.432,A -85,B 0,C 180,E1 -13745.903,E2 -13745.903} C_VEL
LIN {X 0,Y 355.737,Z 434.981,A -85,B 0,C 180,E1 -13746.554,E2 -13746.554} C_VEL
LIN {X 0,Y 359.346,Z 453.896,A -85,B 0,C 180,E1 -13747.269,E2 -13747.269} C_VEL
LIN {X 0,Y 357.851,Z 526.689,A -85,B 0,C 180,E1 -13748.771,E2 -13748.771} C_VEL
LIN {X 0,Y 357.207,Z 539.662,A -85,B 0,C 180,E1 -13749.222,E2 -13749.222} C_VEL
LIN {X 0,Y 356.14,Z 552.156,A -85,B 0,C 180,E1 -13749.873,E2 -13749.873} C_VEL
LIN {X 0,Y 354.923,Z 564.675,A -85,B 0,C 180,E1 -13750.781,E2 -13750.781} C_VEL
LIN {X 0,Y 353.682,Z 575.121,A -85,B 0,C 180,E1 -13751.763,E2 -13751.763} C_VEL
LIN {X 0,Y 352.133,Z 586.182,A -85,B 0,C 180,E1 -13753.074,E2 -13753.074} C_VEL
LIN {X 0,Y 350.916,Z 595.37,A -85,B 0,C 180,E1 -13754.436,E2 -13754.436} C_VEL
LIN {X 0,Y 349.625,Z 604.208,A -85,B 0,C 180,E1 -13756.042,E2 -13756.042} C_VEL
LIN {X 0,Y 348.384,Z 611.843,A -85,B 0,C 180,E1 -13757.772,E2 -13757.772} C_VEL
LIN {X 0,Y 347.559,Z 617.99,A -85,B 0,C 180,E1 -13759.515,E2 -13759.515} C_VEL
LIN {X 0,Y 346.878,Z 622.888,A -85,B 0,C 180,E1 -13761.26,E2 -13761.26} C_VEL
LIN {X 0,Y 346.444,Z 626.678,A -85,B 0,C 180,E1 -13763.009,E2 -13763.009} C_VEL
LIN {X 0,Y 346.214,Z 630.191,A -85,B 0,C 180,E1 -13765.343,E2 -13765.343} C_VEL
LIN {X 0,Y 346.13,Z 631.312,A -85,B 0,C 180,E1 -13766.508,E2 -13766.508} C_VEL
LIN {X 0,Y 346.051,Z 632.348,A -85,B 0,C 180,E1 -13768.837,E2 -13768.837} C_VEL
LIN {X 0,Y 346.091,Z 632.293,A -85,B 0,C 180,E1 -13770,E2 -13770} C_VEL
LIN {X 0,Y 346.053,Z 631.829,A -85,B 0,C 180,E1 -13771.164,E2 -13771.164} C_VEL
LIN {X 0,Y 346.124,Z 629.656,A -85,B 0,C 180,E1 -13773.493,E2 -13773.493} C_VEL
LIN {X 0,Y 346.171,Z 626.52,A -85,B 0,C 180,E1 -13775.46,E2 -13775.46} C_VEL
LIN {X 0,Y 346.48,Z 621.668,A -85,B 0,C 180,E1 -13777.576,E2 -13777.576} C_VEL
LIN {X 0,Y 346.944,Z 615.331,A -85,B 0,C 180,E1 -13779.62,E2 -13779.62} C_VEL
LIN {X 0,Y 347.551,Z 608.416,A -85,B 0,C 180,E1 -13781.371,E2 -13781.371} C_VEL
LIN {X 0,Y 348.495,Z 599.755,A -85,B 0,C 180,E1 -13783.113,E2 -13783.113} C_VEL
LIN {X 0,Y 349.412,Z 590.846,A -85,B 0,C 180,E1 -13784.562,E2 -13784.562} C_VEL
LIN {X 0,Y 350.299,Z 580.898,A -85,B 0,C 180,E1 -13785.882,E2 -13785.882} C_VEL
LIN {X 0,Y 351.251,Z 570.286,A -85,B 0,C 180,E1 -13787.015,E2 -13787.015} C_VEL
LIN {X 0,Y 352.26,Z 558.211,A -85,B 0,C 180,E1 -13788.014,E2 -13788.014} C_VEL
LIN {X 0,Y 353.091,Z 545.6,A -85,B 0,C 180,E1 -13788.796,E2 -13788.796} C_VEL
LIN {X 0,Y 353.759,Z 533.433,A -85,B 0,C 180,E1 -13789.324,E2 -13789.324} C_VEL
LIN {X 0,Y 354.121,Z 519.816,A -85,B 0,C 180,E1 -13789.68,E2 -13789.68} C_VEL
LIN {X 0,Y 355.071,Z 452.144,A -85,B 0,C 180,E1 -13791.048,E2 -13791.048} C_VEL
LIN {X 0,Y 350.283,Z 420.834,A -85,B 0,C 180,E1 -13791.979,E2 -13791.979} C_VEL
LIN {X 0,Y 350.514,Z 417.427,A -85,B 0,C 180,E1 -13792.731,E2 -13792.731} C_VEL
LIN {X 0,Y 350.967,Z 412.653,A -85,B 0,C 180,E1 -13793.922,E2 -13793.922} C_VEL
LIN {X 0,Y 349.269,Z 402.7,A -85,B 0,C 180,E1 -13796.597,E2 -13796.597} C_VEL
LIN {X 0,Y 347.876,Z 395.691,A -85,B 0,C 180,E1 -13798.611,E2 -13798.611} C_VEL
LIN {X 0,Y 347.733,Z 395.668,A -85,B 0,C 180,E1 -13803.072,E2 -13803.072} C_VEL
LIN {X 0,Y 347.772,Z 395.663,A -85,B 0,C 180,E1 -13806.065,E2 -13806.065} C_VEL
LIN {X 0,Y 347.753,Z 395.664,A -85,B 0,C 180,E1 -13808.792,E2 -13808.792} C_VEL
LIN {X 0,Y 347.751,Z 395.667,A -85,B 0,C 180,E1 -13811.83,E2 -13811.83} C_VEL
LIN {X 0,Y 347.796,Z 395.659,A -85,B 0,C 180,E1 -13815.011,E2 -13815.011} C_VEL
LIN {X 0,Y 347.782,Z 395.66,A -85,B 0,C 180,E1 -13818.39,E2 -13818.39} C_VEL
LIN {X 0,Y 347.774,Z 395.662,A -85,B 0,C 180,E1 -13822.01,E2 -13822.01} C_VEL
LIN {X 0,Y 347.742,Z 395.671,A -85,B 0,C 180,E1 -13825.536,E2 -13825.536} C_VEL
LIN {X 0,Y 347.761,Z 395.666,A -85,B 0,C 180,E1 -13829.653,E2 -13829.653} C_VEL
LIN {X 0,Y 347.848,Z 395.652,A -85,B 0,C 180,E1 -13832.744,E2 -13832.744} C_VEL
LIN {X 0,Y 347.782,Z 395.661,A -85,B 0,C 180,E1 -13836.161,E2 -13836.161} C_VEL
LIN {X 0,Y 347.807,Z 395.657,A -85,B 0,C 180,E1 -13839.909,E2 -13839.909} C_VEL
LIN {X 0,Y 347.862,Z 395.65,A -85,B 0,C 180,E1 -13842.359,E2 -13842.359} C_VEL
LIN {X 0,Y 347.893,Z 395.647,A -85,B 0,C 180,E1 -13845.97,E2 -13845.97} C_VEL
LIN {X 0,Y 347.923,Z 395.645,A -85,B 0,C 180,E1 -13849.525,E2 -13849.525} C_VEL
LIN {X 0,Y 348.087,Z 395.625,A -85,B 0,C 180,E1 -13853.042,E2 -13853.042} C_VEL
LIN {X 0,Y 348.203,Z 395.61,A -85,B 0,C 180,E1 -13857.686,E2 -13857.686} C_VEL
LIN {X 0,Y 348.341,Z 395.589,A -85,B 0,C 180,E1 -13860,E2 -13860} C_VEL
LIN {X 0,Y 348.203,Z 395.607,A -85,B 0,C 180,E1 -13862.313,E2 -13862.313} C_VEL
LIN {X 0,Y 348.088,Z 395.625,A -85,B 0,C 180,E1 -13866.958,E2 -13866.958} C_VEL
LIN {X 0,Y 347.923,Z 395.642,A -85,B 0,C 180,E1 -13870.474,E2 -13870.474} C_VEL
LIN {X 0,Y 347.894,Z 395.645,A -85,B 0,C 180,E1 -13874.15,E2 -13874.15} C_VEL
LIN {X 0,Y 347.886,Z 395.647,A -85,B 0,C 180,E1 -13878.29,E2 -13878.29} C_VEL
LIN {X 0,Y 347.784,Z 395.661,A -85,B 0,C 180,E1 -13881.635,E2 -13881.635} C_VEL
LIN {X 0,Y 347.809,Z 395.661,A -85,B 0,C 180,E1 -13885.109,E2 -13885.109} C_VEL
LIN {X 0,Y 347.809,Z 395.658,A -85,B 0,C 180,E1 -13887.694,E2 -13887.694} C_VEL
LIN {X 0,Y 347.761,Z 395.663,A -85,B 0,C 180,E1 -13890.347,E2 -13890.347} C_VEL
LIN {X 0,Y 347.741,Z 395.665,A -85,B 0,C 180,E1 -13894.464,E2 -13894.464} C_VEL
LIN {X 0,Y 347.771,Z 395.662,A -85,B 0,C 180,E1 -13897.989,E2 -13897.989} C_VEL
LIN {X 0,Y 347.748,Z 395.664,A -85,B 0,C 180,E1 -13901.831,E2 -13901.831} C_VEL
LIN {X 0,Y 347.765,Z 395.668,A -85,B 0,C 180,E1 -13905.017,E2 -13905.017} C_VEL
LIN {X 0,Y 347.766,Z 395.663,A -85,B 0,C 180,E1 -13908.394,E2 -13908.394} C_VEL
LIN {X 0,Y 347.775,Z 395.661,A -85,B 0,C 180,E1 -13912.011,E2 -13912.011} C_VEL
LIN {X 0,Y 347.744,Z 395.665,A -85,B 0,C 180,E1 -13915.537,E2 -13915.537} C_VEL
LIN {X 0,Y 347.764,Z 395.663,A -85,B 0,C 180,E1 -13919.654,E2 -13919.654} C_VEL
LIN {X 0,Y 347.851,Z 395.656,A -85,B 0,C 180,E1 -13922.745,E2 -13922.745} C_VEL
LIN {X 0,Y 347.789,Z 395.659,A -85,B 0,C 180,E1 -13926.162,E2 -13926.162} C_VEL
LIN {X 0,Y 347.813,Z 395.656,A -85,B 0,C 180,E1 -13929.91,E2 -13929.91} C_VEL
LIN {X 0,Y 347.867,Z 395.649,A -85,B 0,C 180,E1 -13932.359,E2 -13932.359} C_VEL
LIN {X 0,Y 347.966,Z 395.804,A -85,B 0,C 180,E1 -13936.569,E2 -13936.569} C_VEL
LIN {X 0,Y 350.371,Z 408.961,A -85,B 0,C 180,E1 -13940.394,E2 -13940.394} C_VEL
LIN {X 0,Y 350.422,Z 411.604,A -85,B 0,C 180,E1 -13941.058,E2 -13941.058} C_VEL
LIN {X 0,Y 351.792,Z 420.579,A -85,B 0,C 180,E1 -13941.367,E2 -13941.367} C_VEL
LIN {X 0,Y 355.333,Z 440.699,A -85,B 0,C 180,E1 -13941.977,E2 -13941.977} C_VEL
LIN {X 0,Y 353.968,Z 518.607,A -85,B 0,C 180,E1 -13943.566,E2 -13943.566} C_VEL
LIN {X 0,Y 353.47,Z 531.534,A -85,B 0,C 180,E1 -13944.045,E2 -13944.045} C_VEL
LIN {X 0,Y 352.804,Z 543.769,A -85,B 0,C 180,E1 -13944.717,E2 -13944.717} C_VEL
LIN {X 0,Y 351.934,Z 555.237,A -85,B 0,C 180,E1 -13945.562,E2 -13945.562} C_VEL
LIN {X 0,Y 350.853,Z 567.044,A -85,B 0,C 180,E1 -13946.698,E2 -13946.698} C_VEL
LIN {X 0,Y 349.801,Z 577.604,A -85,B 0,C 180,E1 -13947.985,E2 -13947.985} C_VEL
LIN {X 0,Y 348.842,Z 587.121,A -85,B 0,C 180,E1 -13949.423,E2 -13949.423} C_VEL
LIN {X 0,Y 348.06,Z 594.912,A -85,B 0,C 180,E1 -13950.867,E2 -13950.867} C_VEL
LIN {X 0,Y 347.356,Z 602.523,A -85,B 0,C 180,E1 -13952.609,E2 -13952.609} C_VEL
LIN {X 0,Y 346.688,Z 609.568,A -85,B 0,C 180,E1 -13954.651,E2 -13954.651} C_VEL
LIN {X 0,Y 346.478,Z 614.022,A -85,B 0,C 180,E1 -13956.321,E2 -13956.321} C_VEL
LIN {X 0,Y 346.193,Z 617.799,A -85,B 0,C 180,E1 -13958.169,E2 -13958.169} C_VEL
LIN {X 0,Y 346.056,Z 619.608,A -85,B 0,C 180,E1 -13959.35,E2 -13959.35} C_VEL
LIN {X 0,Y 345.977,Z 620.97,A -85,B 0,C 180,E1 -13960.534,E2 -13960.534} C_VEL
LIN {X 0,Y 346.021,Z 622.475,A -85,B 0,C 180,E1 -13962.858,E2 -13962.858} C_VEL
LIN {X 0,Y 345.891,Z 622.603,A -85,B 0,C 180,E1 -13964.112,E2 -13964.112} C_VEL
LIN {X 0,Y 345.913,Z 622.305,A -85,B 0,C 180,E1 -13965.314,E2 -13965.314} C_VEL
LIN {X 0,Y 346.161,Z 620.805,A -85,B 0,C 180,E1 -13967.403,E2 -13967.403} C_VEL
LIN {X 0,Y 346.509,Z 617.902,A -85,B 0,C 180,E1 -13969.551,E2 -13969.551} C_VEL
LIN {X 0,Y 346.996,Z 614.25,A -85,B 0,C 180,E1 -13971.38,E2 -13971.38} C_VEL
LIN {X 0,Y 347.646,Z 609.385,A -85,B 0,C 180,E1 -13973.216,E2 -13973.216} C_VEL
LIN {X 0,Y 348.593,Z 603.155,A -85,B 0,C 180,E1 -13975.047,E2 -13975.047} C_VEL
LIN {X 0,Y 349.791,Z 595.321,A -85,B 0,C 180,E1 -13976.876,E2 -13976.876} C_VEL
LIN {X 0,Y 351.119,Z 586.491,A -85,B 0,C 180,E1 -13978.512,E2 -13978.512} C_VEL
LIN {X 0,Y 352.591,Z 576.091,A -85,B 0,C 180,E1 -13980.052,E2 -13980.052} C_VEL
LIN {X 0,Y 353.968,Z 565.906,A -85,B 0,C 180,E1 -13981.257,E2 -13981.257} C_VEL
LIN {X 0,Y 354.526,Z 560.916,A -85,B 0,C 180,E1 -13981.76,E2 -13981.76} C_VEL
LIN {X 0,Y 354.461,Z 555.019,A -85,B 0,C 180,E1 -13982.337,E2 -13982.337} C_VEL
LIN {X 0,Y 352.803,Z 547.569,A -85,B 0,C 180,E1 -13983.09,E2 -13983.09} C_VEL
LIN {X 0,Y 350.903,Z 538.993,A -85,B 0,C 180,E1 -13983.834,E2 -13983.834} C_VEL
LIN {X 0,Y 350.644,Z 533.472,A -85,B 0,C 180,E1 -13984.168,E2 -13984.168} C_VEL
LIN {X 0,Y 351.442,Z 520.418,A -85,B 0,C 180,E1 -13984.678,E2 -13984.678} C_VEL
LIN {X 0,Y 352.291,Z 488.357,A -85,B 0,C 180,E1 -13985.377,E2 -13985.377} C_VEL
LIN {X 0,Y 353.274,Z 442.968,A -85,B 0,C 180,E1 -13986.321,E2 -13986.321} C_VEL
LIN {X 0,Y 348.992,Z 423.533,A -85,B 0,C 180,E1 -13987.132,E2 -13987.132} C_VEL
LIN {X 0,Y 344.172,Z 412.172,A -85,B 0,C 180,E1 -13987.862,E2 -13987.862} C_VEL
LIN {X 0,Y 342.774,Z 405.257,A -85,B 0,C 180,E1 -13989.995,E2 -13989.995} C_VEL
LIN {X 0,Y 340.773,Z 396.58,A -85,B 0,C 180,E1 -13993.023,E2 -13993.023} C_VEL
LIN {X 0,Y 340.774,Z 396.537,A -85,B 0,C 180,E1 -13996.204,E2 -13996.204} C_VEL
LIN {X 0,Y 340.759,Z 396.539,A -85,B 0,C 180,E1 -13999.737,E2 -13999.737} C_VEL
LIN {X 0,Y 340.705,Z 396.545,A -85,B 0,C 180,E1 -14003.558,E2 -14003.558} C_VEL
LIN {X 0,Y 340.689,Z 396.538,A -85,B 0,C 180,E1 -14006.153,E2 -14006.153} C_VEL
LIN {X 0,Y 340.769,Z 396.517,A -85,B 0,C 180,E1 -14010.332,E2 -14010.332} C_VEL
LIN {X 0,Y 340.798,Z 396.537,A -85,B 0,C 180,E1 -14013.02,E2 -14013.02} C_VEL
LIN {X 0,Y 340.725,Z 396.542,A -85,B 0,C 180,E1 -14016.927,E2 -14016.927} C_VEL
LIN {X 0,Y 340.794,Z 396.532,A -85,B 0,C 180,E1 -14020.734,E2 -14020.734} C_VEL
LIN {X 0,Y 340.78,Z 396.538,A -85,B 0,C 180,E1 -14023.218,E2 -14023.218} C_VEL
LIN {X 0,Y 340.839,Z 396.527,A -85,B 0,C 180,E1 -14026.89,E2 -14026.89} C_VEL
LIN {X 0,Y 340.922,Z 396.51,A -85,B 0,C 180,E1 -14030.508,E2 -14030.508} C_VEL
LIN {X 0,Y 341.068,Z 396.498,A -85,B 0,C 180,E1 -14032.898,E2 -14032.898} C_VEL
LIN {X 0,Y 341.171,Z 396.483,A -85,B 0,C 180,E1 -14037.639,E2 -14037.639} C_VEL
LIN {X 0,Y 341.309,Z 396.463,A -85,B 0,C 180,E1 -14040,E2 -14040} C_VEL
LIN {X 0,Y 341.163,Z 396.488,A -85,B 0,C 180,E1 -14042.361,E2 -14042.361} C_VEL
LIN {X 0,Y 341.068,Z 396.498,A -85,B 0,C 180,E1 -14047.102,E2 -14047.102} C_VEL
LIN {X 0,Y 340.867,Z 396.525,A -85,B 0,C 180,E1 -14050.694,E2 -14050.694} C_VEL
LIN {X 0,Y 340.856,Z 396.517,A -85,B 0,C 180,E1 -14054.325,E2 -14054.325} C_VEL
LIN {X 0,Y 340.831,Z 396.521,A -85,B 0,C 180,E1 -14058.467,E2 -14058.467} C_VEL
LIN {X 0,Y 340.747,Z 396.535,A -85,B 0,C 180,E1 -14061.858,E2 -14061.858} C_VEL
LIN {X 0,Y 340.766,Z 396.534,A -85,B 0,C 180,E1 -14065.665,E2 -14065.665} C_VEL
LIN {X 0,Y 340.735,Z 396.54,A -85,B 0,C 180,E1 -14068.32,E2 -14068.32} C_VEL
LIN {X 0,Y 340.698,Z 396.542,A -85,B 0,C 180,E1 -14071.045,E2 -14071.045} C_VEL
LIN {X 0,Y 340.713,Z 396.544,A -85,B 0,C 180,E1 -14075.28,E2 -14075.28} C_VEL
LIN {X 0,Y 340.713,Z 396.543,A -85,B 0,C 180,E1 -14078.389,E2 -14078.389} C_VEL
LIN {X 0,Y 340.721,Z 396.523,A -85,B 0,C 180,E1 -14081.305,E2 -14081.305} C_VEL
LIN {X 0,Y 340.734,Z 396.541,A -85,B 0,C 180,E1 -14084.531,E2 -14084.531} C_VEL
LIN {X 0,Y 340.691,Z 396.547,A -85,B 0,C 180,E1 -14088.693,E2 -14088.693} C_VEL
LIN {X 0,Y 340.732,Z 396.543,A -85,B 0,C 180,E1 -14091.774,E2 -14091.774} C_VEL
LIN {X 0,Y 340.721,Z 396.539,A -85,B 0,C 180,E1 -14095.596,E2 -14095.596} C_VEL
LIN {X 0,Y 340.714,Z 396.738,A -85,B 0,C 180,E1 -14098.013,E2 -14098.013} C_VEL
LIN {X 0,Y 343.107,Z 406.411,A -85,B 0,C 180,E1 -14101.196,E2 -14101.196} C_VEL
LIN {X 0,Y 345.147,Z 416.354,A -85,B 0,C 180,E1 -14104.225,E2 -14104.225} C_VEL
LIN {X 0,Y 345.701,Z 420.279,A -85,B 0,C 180,E1 -14105.308,E2 -14105.308} C_VEL
LIN {X 0,Y 347.672,Z 428.615,A -85,B 0,C 180,E1 -14105.721,E2 -14105.721} C_VEL
LIN {X 0,Y 351.81,Z 448.063,A -85,B 0,C 180,E1 -14106.523,E2 -14106.523} C_VEL
LIN {X 0,Y 353.078,Z 455.66,A -85,B 0,C 180,E1 -14106.801,E2 -14106.801} C_VEL
LIN {X 0,Y 351.361,Z 528.083,A -85,B 0,C 180,E1 -14108.321,E2 -14108.321} C_VEL
LIN {X 0,Y 350.652,Z 541.17,A -85,B 0,C 180,E1 -14108.815,E2 -14108.815} C_VEL
LIN {X 0,Y 349.553,Z 553.249,A -85,B 0,C 180,E1 -14109.477,E2 -14109.477} C_VEL
LIN {X 0,Y 348.27,Z 565.458,A -85,B 0,C 180,E1 -14110.399,E2 -14110.399} C_VEL
LIN {X 0,Y 346.766,Z 576.99,A -85,B 0,C 180,E1 -14111.539,E2 -14111.539} C_VEL
LIN {X 0,Y 345.254,Z 587.383,A -85,B 0,C 180,E1 -14112.833,E2 -14112.833} C_VEL
LIN {X 0,Y 344.075,Z 595.922,A -85,B 0,C 180,E1 -14114.153,E2 -14114.153} C_VEL
LIN {X 0,Y 342.756,Z 604.466,A -85,B 0,C 180,E1 -14115.757,E2 -14115.757} C_VEL
LIN {X 0,Y 341.421,Z 612.021,A -85,B 0,C 180,E1 -14117.518,E2 -14117.518} C_VEL
LIN {X 0,Y 340.548,Z 618.115,A -85,B 0,C 180,E1 -14119.296,E2 -14119.296} C_VEL
LIN {X 0,Y 339.861,Z 622.965,A -85,B 0,C 180,E1 -14121.078,E2 -14121.078} C_VEL
LIN {X 0,Y 339.396,Z 626.71,A -85,B 0,C 180,E1 -14122.863,E2 -14122.863} C_VEL
LIN {X 0,Y 339.21,Z 628.648,A -85,B 0,C 180,E1 -14124.054,E2 -14124.054} C_VEL
LIN {X 0,Y 339.118,Z 630.177,A -85,B 0,C 180,E1 -14125.245,E2 -14125.245} C_VEL
LIN {X 0,Y 339.059,Z 631.262,A -85,B 0,C 180,E1 -14126.435,E2 -14126.435} C_VEL
LIN {X 0,Y 338.957,Z 632.258,A -85,B 0,C 180,E1 -14128.812,E2 -14128.812} C_VEL
LIN {X 0,Y 338.993,Z 632.182,A -85,B 0,C 180,E1 -14130,E2 -14130} C_VEL
LIN {X 0,Y 338.958,Z 631.678,A -85,B 0,C 180,E1 -14131.188,E2 -14131.188} C_VEL
LIN {X 0,Y 339.051,Z 629.464,A -85,B 0,C 180,E1 -14133.565,E2 -14133.565} C_VEL
LIN {X 0,Y 339.068,Z 626.628,A -85,B 0,C 180,E1 -14135.384,E2 -14135.384} C_VEL
LIN {X 0,Y 339.279,Z 622.874,A -85,B 0,C 180,E1 -14137.14,E2 -14137.14} C_VEL
LIN {X 0,Y 339.7,Z 617.925,A -85,B 0,C 180,E1 -14138.927,E2 -14138.927} C_VEL
LIN {X 0,Y 340.256,Z 611.681,A -85,B 0,C 180,E1 -14140.713,E2 -14140.713} C_VEL
LIN {X 0,Y 341.039,Z 603.87,A -85,B 0,C 180,E1 -14142.497,E2 -14142.497} C_VEL
LIN {X 0,Y 341.833,Z 595.864,A -85,B 0,C 180,E1 -14143.98,E2 -14143.98} C_VEL
LIN {X 0,Y 342.872,Z 586.086,A -85,B 0,C 180,E1 -14145.454,E2 -14145.454} C_VEL
LIN {X 0,Y 343.87,Z 575.193,A -85,B 0,C 180,E1 -14146.779,E2 -14146.779} C_VEL
LIN {X 0,Y 344.832,Z 564.548,A -85,B 0,C 180,E1 -14147.801,E2 -14147.801} C_VEL
LIN {X 0,Y 345.868,Z 551.716,A -85,B 0,C 180,E1 -14148.742,E2 -14148.742} C_VEL
LIN {X 0,Y 346.674,Z 538.812,A -85,B 0,C 180,E1 -14149.426,E2 -14149.426} C_VEL
LIN {X 0,Y 347.202,Z 526.149,A -85,B 0,C 180,E1 -14149.857,E2 -14149.857} C_VEL
LIN {X 0,Y 348.333,Z 453.251,A -85,B 0,C 180,E1 -14151.372,E2 -14151.372} C_VEL
LIN {X 0,Y 343.435,Z 420.771,A -85,B 0,C 180,E1 -14152.356,E2 -14152.356} C_VEL
LIN {X 0,Y 343.532,Z 418.332,A -85,B 0,C 180,E1 -14152.874,E2 -14152.874} C_VEL
LIN {X 0,Y 343.952,Z 413.449,A -85,B 0,C 180,E1 -14154.121,E2 -14154.121} C_VEL
LIN {X 0,Y 341.904,Z 401.858,A -85,B 0,C 180,E1 -14157.317,E2 -14157.317} C_VEL
LIN {X 0,Y 340.829,Z 396.586,A -85,B 0,C 180,E1 -14158.879,E2 -14158.879} C_VEL
LIN {X 0,Y 340.686,Z 396.545,A -85,B 0,C 180,E1 -14162.435,E2 -14162.435} C_VEL
LIN {X 0,Y 340.719,Z 396.543,A -85,B 0,C 180,E1 -14165.278,E2 -14165.278} C_VEL
LIN {X 0,Y 340.712,Z 396.54,A -85,B 0,C 180,E1 -14168.386,E2 -14168.386} C_VEL
LIN {X 0,Y 340.699,Z 396.544,A -85,B 0,C 180,E1 -14172.045,E2 -14172.045} C_VEL
LIN {X 0,Y 340.719,Z 396.541,A -85,B 0,C 180,E1 -14175.467,E2 -14175.467} C_VEL
LIN {X 0,Y 340.723,Z 396.539,A -85,B 0,C 180,E1 -14178.696,E2 -14178.696} C_VEL
LIN {X 0,Y 340.737,Z 396.541,A -85,B 0,C 180,E1 -14181.773,E2 -14181.773} C_VEL
LIN {X 0,Y 340.72,Z 396.545,A -85,B 0,C 180,E1 -14185.595,E2 -14185.595} C_VEL
LIN {X 0,Y 340.701,Z 396.544,A -85,B 0,C 180,E1 -14188.955,E2 -14188.955} C_VEL
LIN {X 0,Y 340.775,Z 396.532,A -85,B 0,C 180,E1 -14192.474,E2 -14192.474} C_VEL
LIN {X 0,Y 340.751,Z 396.54,A -85,B 0,C 180,E1 -14195.638,E2 -14195.638} C_VEL
LIN {X 0,Y 340.734,Z 396.541,A -85,B 0,C 180,E1 -14199.473,E2 -14199.473} C_VEL
LIN {X 0,Y 340.854,Z 396.524,A -85,B 0,C 180,E1 -14201.984,E2 -14201.984} C_VEL
LIN {X 0,Y 340.865,Z 396.524,A -85,B 0,C 180,E1 -14205.705,E2 -14205.705} C_VEL
LIN {X 0,Y 340.866,Z 396.525,A -85,B 0,C 180,E1 -14209.306,E2 -14209.306} C_VEL
LIN {X 0,Y 341.055,Z 396.5,A -85,B 0,C 180,E1 -14212.898,E2 -14212.898} C_VEL
LIN {X 0,Y 341.165,Z 396.486,A -85,B 0,C 180,E1 -14217.639,E2 -14217.639} C_VEL
LIN {X 0,Y 341.291,Z 396.466,A -85,B 0,C 180,E1 -14220,E2 -14220} C_VEL
LIN {X 0,Y 341.165,Z 396.482,A -85,B 0,C 180,E1 -14222.361,E2 -14222.361} C_VEL
LIN {X 0,Y 341.056,Z 396.503,A -85,B 0,C 180,E1 -14227.102,E2 -14227.102} C_VEL
LIN {X 0,Y 340.866,Z 396.522,A -85,B 0,C 180,E1 -14230.694,E2 -14230.694} C_VEL
LIN {X 0,Y 340.859,Z 396.521,A -85,B 0,C 180,E1 -14234.325,E2 -14234.325} C_VEL
LIN {X 0,Y 340.833,Z 396.526,A -85,B 0,C 180,E1 -14238.466,E2 -14238.466} C_VEL
LIN {X 0,Y 340.75,Z 396.535,A -85,B 0,C 180,E1 -14241.857,E2 -14241.857} C_VEL
LIN {X 0,Y 340.769,Z 396.534,A -85,B 0,C 180,E1 -14245.665,E2 -14245.665} C_VEL
LIN {X 0,Y 340.739,Z 396.538,A -85,B 0,C 180,E1 -14248.32,E2 -14248.32} C_VEL
LIN {X 0,Y 340.701,Z 396.547,A -85,B 0,C 180,E1 -14251.044,E2 -14251.044} C_VEL
LIN {X 0,Y 340.715,Z 396.545,A -85,B 0,C 180,E1 -14255.279,E2 -14255.279} C_VEL
LIN {X 0,Y 340.707,Z 396.542,A -85,B 0,C 180,E1 -14258.386,E2 -14258.386} C_VEL
LIN {X 0,Y 340.697,Z 396.541,A -85,B 0,C 180,E1 -14262.046,E2 -14262.046} C_VEL
LIN {X 0,Y 340.687,Z 396.547,A -85,B 0,C 180,E1 -14265.463,E2 -14265.463} C_VEL
LIN {X 0,Y 340.703,Z 396.544,A -85,B 0,C 180,E1 -14268.694,E2 -14268.694} C_VEL
LIN {X 0,Y 340.738,Z 396.539,A -85,B 0,C 180,E1 -14271.774,E2 -14271.774} C_VEL
LIN {X 0,Y 340.722,Z 396.538,A -85,B 0,C 180,E1 -14275.596,E2 -14275.596} C_VEL
LIN {X 0,Y 340.703,Z 396.544,A -85,B 0,C 180,E1 -14278.956,E2 -14278.956} C_VEL
LIN {X 0,Y 340.778,Z 396.535,A -85,B 0,C 180,E1 -14282.475,E2 -14282.475} C_VEL
LIN {X 0,Y 340.756,Z 396.535,A -85,B 0,C 180,E1 -14285.639,E2 -14285.639} C_VEL
LIN {X 0,Y 340.753,Z 396.536,A -85,B 0,C 180,E1 -14289.475,E2 -14289.475} C_VEL
LIN {X 0,Y 340.858,Z 396.52,A -85,B 0,C 180,E1 -14291.984,E2 -14291.984} C_VEL
LIN {X 0,Y 340.92,Z 396.717,A -85,B 0,C 180,E1 -14296.324,E2 -14296.324} C_VEL
LIN {X 0,Y 343.144,Z 408.764,A -85,B 0,C 180,E1 -14299.901,E2 -14299.901} C_VEL
LIN {X 0,Y 343.49,Z 411.932,A -85,B 0,C 180,E1 -14300.701,E2 -14300.701} C_VEL
LIN {X 0,Y 347.092,Z 432.596,A -85,B 0,C 180,E1 -14301.373,E2 -14301.373} C_VEL
LIN {X 0,Y 348.57,Z 441.846,A -85,B 0,C 180,E1 -14301.649,E2 -14301.649} C_VEL
LIN {X 0,Y 347.15,Z 518.643,A -85,B 0,C 180,E1 -14303.243,E2 -14303.243} C_VEL
LIN {X 0,Y 346.631,Z 531.832,A -85,B 0,C 180,E1 -14303.743,E2 -14303.743} C_VEL
LIN {X 0,Y 345.899,Z 544.543,A -85,B 0,C 180,E1 -14304.461,E2 -14304.461} C_VEL
LIN {X 0,Y 345.012,Z 555.891,A -85,B 0,C 180,E1 -14305.326,E2 -14305.326} C_VEL
LIN {X 0,Y 343.883,Z 567.572,A -85,B 0,C 180,E1 -14306.485,E2 -14306.485} C_VEL
LIN {X 0,Y 342.812,Z 578.057,A -85,B 0,C 180,E1 -14307.797,E2 -14307.797} C_VEL
LIN {X 0,Y 341.889,Z 586.631,A -85,B 0,C 180,E1 -14309.116,E2 -14309.116} C_VEL
LIN {X 0,Y 341.115,Z 594.524,A -85,B 0,C 180,E1 -14310.59,E2 -14310.59} C_VEL
LIN {X 0,Y 340.341,Z 602.248,A -85,B 0,C 180,E1 -14312.367,E2 -14312.367} C_VEL
LIN {X 0,Y 339.677,Z 608.457,A -85,B 0,C 180,E1 -14314.152,E2 -14314.152} C_VEL
LIN {X 0,Y 339.402,Z 614.262,A -85,B 0,C 180,E1 -14316.313,E2 -14316.313} C_VEL
LIN {X 0,Y 339.063,Z 618.237,A -85,B 0,C 180,E1 -14318.342,E2 -14318.342} C_VEL
LIN {X 0,Y 338.952,Z 619.954,A -85,B 0,C 180,E1 -14319.548,E2 -14319.548} C_VEL
LIN {X 0,Y 338.868,Z 621.262,A -85,B 0,C 180,E1 -14320.757,E2 -14320.757} C_VEL
LIN {X 0,Y 338.906,Z 622.575,A -85,B 0,C 180,E1 -14322.927,E2 -14322.927} C_VEL
LIN {X 0,Y 338.784,Z 622.678,A -85,B 0,C 180,E1 -14324.414,E2 -14324.414} C_VEL
LIN {X 0,Y 338.832,Z 622.324,A -85,B 0,C 180,E1 -14325.642,E2 -14325.642} C_VEL
LIN {X 0,Y 339.103,Z 620.907,A -85,B 0,C 180,E1 -14327.568,E2 -14327.568} C_VEL
LIN {X 0,Y 339.535,Z 617.634,A -85,B 0,C 180,E1 -14329.969,E2 -14329.969} C_VEL
LIN {X 0,Y 340.062,Z 613.854,A -85,B 0,C 180,E1 -14331.838,E2 -14331.838} C_VEL
LIN {X 0,Y 340.806,Z 608.853,A -85,B 0,C 180,E1 -14333.71,E2 -14333.71} C_VEL
LIN {X 0,Y 341.829,Z 602.477,A -85,B 0,C 180,E1 -14335.578,E2 -14335.578} C_VEL
LIN {X 0,Y 343.138,Z 594.431,A -85,B 0,C 180,E1 -14337.44,E2 -14337.44} C_VEL
LIN {X 0,Y 344.547,Z 585.591,A -85,B 0,C 180,E1 -14339.067,E2 -14339.067} C_VEL
LIN {X 0,Y 345.99,Z 575.848,A -85,B 0,C 180,E1 -14340.518,E2 -14340.518} C_VEL
LIN {X 0,Y 347.414,Z 565.69,A -85,B 0,C 180,E1 -14341.732,E2 -14341.732} C_VEL
LIN {X 0,Y 348.795,Z 553.659,A -85,B 0,C 180,E1 -14342.863,E2 -14342.863} C_VEL
LIN {X 0,Y 350.045,Z 540.871,A -85,B 0,C 180,E1 -14343.771,E2 -14343.771} C_VEL
LIN {X 0,Y 350.644,Z 533.472,A -85,B 0,C 180,E1 -14344.168,E2 -14344.168} C_VEL
LIN {X 0,Y 350.269,Z 529.716,A -85,B 0,C 180,E1 -14344.393,E2 -14344.393} C_VEL
LIN {X 0,Y 345.744,Z 517.995,A -85,B 0,C 180,E1 -14345.213,E2 -14345.213} C_VEL
LIN {X 0,Y 345.32,Z 514.141,A -85,B 0,C 180,E1 -14345.351,E2 -14345.351} C_VEL
LIN {X 0,Y 346.946,Z 444.036,A -85,B 0,C 180,E1 -14346.836,E2 -14346.836} C_VEL
LIN {X 0,Y 342.996,Z 426.005,A -85,B 0,C 180,E1 -14347.608,E2 -14347.608} C_VEL
LIN {X 0,Y 337.041,Z 412.303,A -85,B 0,C 180,E1 -14348.536,E2 -14348.536} C_VEL
LIN {X 0,Y 336.448,Z 409.367,A -85,B 0,C 180,E1 -14349.386,E2 -14349.386} C_VEL
LIN {X 0,Y 334.072,Z 398.933,A -85,B 0,C 180,E1 -14352.986,E2 -14352.986} C_VEL
LIN {X 0,Y 333.735,Z 397.432,A -85,B 0,C 180,E1 -14353.626,E2 -14353.626} C_VEL
LIN {X 0,Y 333.698,Z 397.411,A -85,B 0,C 180,E1 -14357.486,E2 -14357.486} C_VEL
LIN {X 0,Y 333.677,Z 397.411,A -85,B 0,C 180,E1 -14361.195,E2 -14361.195} C_VEL
LIN {X 0,Y 333.68,Z 397.406,A -85,B 0,C 180,E1 -14365.225,E2 -14365.225} C_VEL
LIN {X 0,Y 333.638,Z 397.425,A -85,B 0,C 180,E1 -14368.223,E2 -14368.223} C_VEL
LIN {X 0,Y 333.705,Z 397.4,A -85,B 0,C 180,E1 -14371.027,E2 -14371.027} C_VEL
LIN {X 0,Y 333.729,Z 397.413,A -85,B 0,C 180,E1 -14373.753,E2 -14373.753} C_VEL
LIN {X 0,Y 333.713,Z 397.408,A -85,B 0,C 180,E1 -14377.913,E2 -14377.913} C_VEL
LIN {X 0,Y 333.788,Z 397.399,A -85,B 0,C 180,E1 -14381.589,E2 -14381.589} C_VEL
LIN {X 0,Y 333.801,Z 397.397,A -85,B 0,C 180,E1 -14385.576,E2 -14385.576} C_VEL
LIN {X 0,Y 333.83,Z 397.394,A -85,B 0,C 180,E1 -14389.078,E2 -14389.078} C_VEL
LIN {X 0,Y 334.017,Z 397.378,A -85,B 0,C 180,E1 -14392.747,E2 -14392.747} C_VEL
LIN {X 0,Y 334.133,Z 397.36,A -85,B 0,C 180,E1 -14397.589,E2 -14397.589} C_VEL
LIN {X 0,Y 334.259,Z 397.341,A -85,B 0,C 180,E1 -14400,E2 -14400} C_VEL
LIN {X 0,Y 334.124,Z 397.365,A -85,B 0,C 180,E1 -14402.411,E2 -14402.411} C_VEL
LIN {X 0,Y 334.017,Z 397.375,A -85,B 0,C 180,E1 -14407.253,E2 -14407.253} C_VEL
LIN {X 0,Y 333.83,Z 397.404,A -85,B 0,C 180,E1 -14410.922,E2 -14410.922} C_VEL
LIN {X 0,Y 333.801,Z 397.398,A -85,B 0,C 180,E1 -14414.635,E2 -14414.635} C_VEL
LIN {X 0,Y 333.79,Z 397.398,A -85,B 0,C 180,E1 -14418.656,E2 -14418.656} C_VEL
LIN {X 0,Y 333.686,Z 397.413,A -85,B 0,C 180,E1 -14422.279,E2 -14422.279} C_VEL
LIN {X 0,Y 333.729,Z 397.409,A -85,B 0,C 180,E1 -14426.247,E2 -14426.247} C_VEL
LIN {X 0,Y 333.705,Z 397.417,A -85,B 0,C 180,E1 -14428.973,E2 -14428.973} C_VEL
LIN {X 0,Y 333.637,Z 397.428,A -85,B 0,C 180,E1 -14432.588,E2 -14432.588} C_VEL
LIN {X 0,Y 333.672,Z 397.423,A -85,B 0,C 180,E1 -14436.14,E2 -14436.14} C_VEL
LIN {X 0,Y 333.68,Z 397.419,A -85,B 0,C 180,E1 -14439.188,E2 -14439.188} C_VEL
LIN {X 0,Y 333.686,Z 397.404,A -85,B 0,C 180,E1 -14442.512,E2 -14442.512} C_VEL
LIN {X 0,Y 333.631,Z 397.414,A -85,B 0,C 180,E1 -14445.962,E2 -14445.962} C_VEL
LIN {X 0,Y 333.649,Z 397.419,A -85,B 0,C 180,E1 -14449.315,E2 -14449.315} C_VEL
LIN {X 0,Y 333.663,Z 397.414,A -85,B 0,C 180,E1 -14453.169,E2 -14453.169} C_VEL
LIN {X 0,Y 333.672,Z 397.419,A -85,B 0,C 180,E1 -14455.342,E2 -14455.342} C_VEL
LIN {X 0,Y 333.672,Z 397.565,A -85,B 0,C 180,E1 -14457.406,E2 -14457.406} C_VEL
LIN {X 0,Y 335.647,Z 405.674,A -85,B 0,C 180,E1 -14460.18,E2 -14460.18} C_VEL
LIN {X 0,Y 337.78,Z 415.168,A -85,B 0,C 180,E1 -14463.197,E2 -14463.197} C_VEL
LIN {X 0,Y 338.661,Z 420.093,A -85,B 0,C 180,E1 -14464.643,E2 -14464.643} C_VEL
LIN {X 0,Y 340.196,Z 424.677,A -85,B 0,C 180,E1 -14464.953,E2 -14464.953} C_VEL
LIN {X 0,Y 345.133,Z 447.202,A -85,B 0,C 180,E1 -14465.93,E2 -14465.93} C_VEL
LIN {X 0,Y 346.741,Z 457.157,A -85,B 0,C 180,E1 -14466.301,E2 -14466.301} C_VEL
LIN {X 0,Y 344.971,Z 528.134,A -85,B 0,C 180,E1 -14467.82,E2 -14467.82} C_VEL
LIN {X 0,Y 344.209,Z 541.176,A -85,B 0,C 180,E1 -14468.32,E2 -14468.32} C_VEL
LIN {X 0,Y 343.079,Z 553.226,A -85,B 0,C 180,E1 -14468.993,E2 -14468.993} C_VEL
LIN {X 0,Y 341.856,Z 564.593,A -85,B 0,C 180,E1 -14469.858,E2 -14469.858} C_VEL
LIN {X 0,Y 340.279,Z 576.293,A -85,B 0,C 180,E1 -14471.017,E2 -14471.017} C_VEL
LIN {X 0,Y 338.67,Z 586.789,A -85,B 0,C 180,E1 -14472.333,E2 -14472.333} C_VEL
LIN {X 0,Y 337.24,Z 596.503,A -85,B 0,C 180,E1 -14473.86,E2 -14473.86} C_VEL
LIN {X 0,Y 335.894,Z 604.728,A -85,B 0,C 180,E1 -14475.459,E2 -14475.459} C_VEL
LIN {X 0,Y 334.487,Z 612.218,A -85,B 0,C 180,E1 -14477.255,E2 -14477.255} C_VEL
LIN {X 0,Y 333.55,Z 618.252,A -85,B 0,C 180,E1 -14479.069,E2 -14479.069} C_VEL
LIN {X 0,Y 332.827,Z 623.048,A -85,B 0,C 180,E1 -14480.888,E2 -14480.888} C_VEL
LIN {X 0,Y 332.346,Z 626.745,A -85,B 0,C 180,E1 -14482.711,E2 -14482.711} C_VEL
LIN {X 0,Y 332.136,Z 628.77,A -85,B 0,C 180,E1 -14484.002,E2 -14484.002} C_VEL
LIN {X 0,Y 332.026,Z 630.156,A -85,B 0,C 180,E1 -14485.143,E2 -14485.143} C_VEL
LIN {X 0,Y 331.967,Z 631.211,A -85,B 0,C 180,E1 -14486.359,E2 -14486.359} C_VEL
LIN {X 0,Y 331.866,Z 632.167,A -85,B 0,C 180,E1 -14488.787,E2 -14488.787} C_VEL
LIN {X 0,Y 331.898,Z 632.064,A -85,B 0,C 180,E1 -14490,E2 -14490} C_VEL
LIN {X 0,Y 331.867,Z 631.527,A -85,B 0,C 180,E1 -14491.214,E2 -14491.214} C_VEL
LIN {X 0,Y 331.886,Z 630.598,A -85,B 0,C 180,E1 -14492.428,E2 -14492.428} C_VEL
LIN {X 0,Y 331.956,Z 629.272,A -85,B 0,C 180,E1 -14493.642,E2 -14493.642} C_VEL
LIN {X 0,Y 332.004,Z 625.892,A -85,B 0,C 180,E1 -14495.777,E2 -14495.777} C_VEL
LIN {X 0,Y 332.368,Z 621.06,A -85,B 0,C 180,E1 -14497.9,E2 -14497.9} C_VEL
LIN {X 0,Y 332.912,Z 614.621,A -85,B 0,C 180,E1 -14500.03,E2 -14500.03} C_VEL
LIN {X 0,Y 333.578,Z 607.571,A -85,B 0,C 180,E1 -14501.854,E2 -14501.854} C_VEL
LIN {X 0,Y 334.609,Z 598.726,A -85,B 0,C 180,E1 -14503.668,E2 -14503.668} C_VEL
LIN {X 0,Y 335.692,Z 588.631,A -85,B 0,C 180,E1 -14505.33,E2 -14505.33} C_VEL
LIN {X 0,Y 336.676,Z 578.334,A -85,B 0,C 180,E1 -14506.68,E2 -14506.68} C_VEL
LIN {X 0,Y 337.756,Z 566.872,A -85,B 0,C 180,E1 -14507.873,E2 -14507.873} C_VEL
LIN {X 0,Y 338.79,Z 554.943,A -85,B 0,C 180,E1 -14508.834,E2 -14508.834} C_VEL
LIN {X 0,Y 339.646,Z 542.479,A -85,B 0,C 180,E1 -14509.57,E2 -14509.57} C_VEL
LIN {X 0,Y 340.302,Z 528.562,A -85,B 0,C 180,E1 -14510.12,E2 -14510.12} C_VEL
LIN {X 0,Y 341.6,Z 454.269,A -85,B 0,C 180,E1 -14511.706,E2 -14511.706} C_VEL
LIN {X 0,Y 336.513,Z 420.522,A -85,B 0,C 180,E1 -14512.767,E2 -14512.767} C_VEL
LIN {X 0,Y 336.935,Z 414.244,A -85,B 0,C 180,E1 -14514.328,E2 -14514.328} C_VEL
LIN {X 0,Y 334.917,Z 402.993,A -85,B 0,C 180,E1 -14517.494,E2 -14517.494} C_VEL
LIN {X 0,Y 333.769,Z 397.448,A -85,B 0,C 180,E1 -14519.182,E2 -14519.182} C_VEL
LIN {X 0,Y 333.637,Z 397.426,A -85,B 0,C 180,E1 -14523.208,E2 -14523.208} C_VEL
LIN {X 0,Y 333.667,Z 397.42,A -85,B 0,C 180,E1 -14526.832,E2 -14526.832} C_VEL
LIN {X 0,Y 333.646,Z 397.421,A -85,B 0,C 180,E1 -14530.767,E2 -14530.767} C_VEL
LIN {X 0,Y 333.641,Z 397.419,A -85,B 0,C 180,E1 -14534.259,E2 -14534.259} C_VEL
LIN {X 0,Y 333.692,Z 397.418,A -85,B 0,C 180,E1 -14537.626,E2 -14537.626} C_VEL
LIN {X 0,Y 333.681,Z 397.42,A -85,B 0,C 180,E1 -14541.195,E2 -14541.195} C_VEL
LIN {X 0,Y 333.683,Z 397.419,A -85,B 0,C 180,E1 -14545.225,E2 -14545.225} C_VEL
LIN {X 0,Y 333.694,Z 397.418,A -85,B 0,C 180,E1 -14549.637,E2 -14549.637} C_VEL
LIN {X 0,Y 333.74,Z 397.408,A -85,B 0,C 180,E1 -14552.401,E2 -14552.401} C_VEL
LIN {X 0,Y 333.722,Z 397.415,A -85,B 0,C 180,E1 -14555.09,E2 -14555.09} C_VEL
LIN {X 0,Y 333.671,Z 397.419,A -85,B 0,C 180,E1 -14559.018,E2 -14559.018} C_VEL
LIN {X 0,Y 333.791,Z 397.406,A -85,B 0,C 180,E1 -14561.589,E2 -14561.589} C_VEL
LIN {X 0,Y 333.804,Z 397.405,A -85,B 0,C 180,E1 -14565.576,E2 -14565.576} C_VEL
LIN {X 0,Y 333.829,Z 397.399,A -85,B 0,C 180,E1 -14569.078,E2 -14569.078} C_VEL
LIN {X 0,Y 334.002,Z 397.377,A -85,B 0,C 180,E1 -14572.747,E2 -14572.747} C_VEL
LIN {X 0,Y 333.806,Z 397.406,A -85,B 0,C 180,E1 -14575.169,E2 -14575.169} C_VEL
LIN {X 0,Y 334.102,Z 397.366,A -85,B 0,C 180,E1 -14577.589,E2 -14577.589} C_VEL
LIN {X 0,Y 334.242,Z 397.343,A -85,B 0,C 180,E1 -14580,E2 -14580} C_VEL
LIN {X 0,Y 334.102,Z 397.361,A -85,B 0,C 180,E1 -14582.411,E2 -14582.411} C_VEL
LIN {X 0,Y 333.988,Z 397.379,A -85,B 0,C 180,E1 -14586.66,E2 -14586.66} C_VEL
LIN {X 0,Y 333.846,Z 397.396,A -85,B 0,C 180,E1 -14589.695,E2 -14589.695} C_VEL
LIN {X 0,Y 333.792,Z 397.405,A -85,B 0,C 180,E1 -14593.392,E2 -14593.392} C_VEL
LIN {X 0,Y 333.742,Z 397.414,A -85,B 0,C 180,E1 -14597.146,E2 -14597.146} C_VEL
LIN {X 0,Y 333.734,Z 397.411,A -85,B 0,C 180,E1 -14599.69,E2 -14599.69} C_VEL
LIN {X 0,Y 333.688,Z 397.413,A -85,B 0,C 180,E1 -14602.278,E2 -14602.278} C_VEL
LIN {X 0,Y 333.732,Z 397.409,A -85,B 0,C 180,E1 -14606.247,E2 -14606.247} C_VEL
LIN {X 0,Y 333.708,Z 397.418,A -85,B 0,C 180,E1 -14608.972,E2 -14608.972} C_VEL
LIN {X 0,Y 333.64,Z 397.421,A -85,B 0,C 180,E1 -14612.587,E2 -14612.587} C_VEL
LIN {X 0,Y 333.673,Z 397.417,A -85,B 0,C 180,E1 -14616.139,E2 -14616.139} C_VEL
LIN {X 0,Y 333.644,Z 397.426,A -85,B 0,C 180,E1 -14619.193,E2 -14619.193} C_VEL
LIN {X 0,Y 333.631,Z 397.421,A -85,B 0,C 180,E1 -14622.5,E2 -14622.5} C_VEL
LIN {X 0,Y 333.631,Z 397.423,A -85,B 0,C 180,E1 -14625.962,E2 -14625.962} C_VEL
LIN {X 0,Y 333.655,Z 397.423,A -85,B 0,C 180,E1 -14629.314,E2 -14629.314} C_VEL
LIN {X 0,Y 333.655,Z 397.421,A -85,B 0,C 180,E1 -14632.35,E2 -14632.35} C_VEL
LIN {X 0,Y 333.673,Z 397.417,A -85,B 0,C 180,E1 -14635.342,E2 -14635.342} C_VEL
LIN {X 0,Y 333.702,Z 397.414,A -85,B 0,C 180,E1 -14639.711,E2 -14639.711} C_VEL
LIN {X 0,Y 333.742,Z 397.411,A -85,B 0,C 180,E1 -14642.401,E2 -14642.401} C_VEL
LIN {X 0,Y 333.727,Z 397.412,A -85,B 0,C 180,E1 -14645.091,E2 -14645.091} C_VEL
LIN {X 0,Y 333.686,Z 397.42,A -85,B 0,C 180,E1 -14649.02,E2 -14649.02} C_VEL
LIN {X 0,Y 333.794,Z 397.4,A -85,B 0,C 180,E1 -14651.59,E2 -14651.59} C_VEL
LIN {X 0,Y 333.819,Z 397.404,A -85,B 0,C 180,E1 -14655.77,E2 -14655.77} C_VEL
LIN {X 0,Y 333.893,Z 397.768,A -85,B 0,C 180,E1 -14656.114,E2 -14656.114} C_VEL
LIN {X 0,Y 335.951,Z 408.934,A -85,B 0,C 180,E1 -14659.492,E2 -14659.492} C_VEL
LIN {X 0,Y 336.436,Z 411.795,A -85,B 0,C 180,E1 -14660.267,E2 -14660.267} C_VEL
LIN {X 0,Y 337.274,Z 415.758,A -85,B 0,C 180,E1 -14660.461,E2 -14660.461} C_VEL
LIN {X 0,Y 340.371,Z 433.888,A -85,B 0,C 180,E1 -14661.034,E2 -14661.034} C_VEL
LIN {X 0,Y 341.777,Z 441.872,A -85,B 0,C 180,E1 -14661.286,E2 -14661.286} C_VEL
LIN {X 0,Y 340.34,Z 518.685,A -85,B 0,C 180,E1 -14662.912,E2 -14662.912} C_VEL
LIN {X 0,Y 339.787,Z 532.293,A -85,B 0,C 180,E1 -14663.44,E2 -14663.44} C_VEL
LIN {X 0,Y 338.996,Z 545.33,A -85,B 0,C 180,E1 -14664.199,E2 -14664.199} C_VEL
LIN {X 0,Y 338.085,Z 556.48,A -85,B 0,C 180,E1 -14665.081,E2 -14665.081} C_VEL
LIN {X 0,Y 336.931,Z 568.07,A -85,B 0,C 180,E1 -14666.262,E2 -14666.262} C_VEL
LIN {X 0,Y 335.825,Z 578.492,A -85,B 0,C 180,E1 -14667.601,E2 -14667.601} C_VEL
LIN {X 0,Y 334.808,Z 587.866,A -85,B 0,C 180,E1 -14669.098,E2 -14669.098} C_VEL
LIN {X 0,Y 333.993,Z 595.556,A -85,B 0,C 180,E1 -14670.603,E2 -14670.603} C_VEL
LIN {X 0,Y 333.25,Z 603.088,A -85,B 0,C 180,E1 -14672.417,E2 -14672.417} C_VEL
LIN {X 0,Y 332.574,Z 609.161,A -85,B 0,C 180,E1 -14674.241,E2 -14674.241} C_VEL
LIN {X 0,Y 332.312,Z 614.449,A -85,B 0,C 180,E1 -14676.282,E2 -14676.282} C_VEL
LIN {X 0,Y 332.054,Z 617.637,A -85,B 0,C 180,E1 -14677.907,E2 -14677.907} C_VEL
LIN {X 0,Y 331.827,Z 620.301,A -85,B 0,C 180,E1 -14679.755,E2 -14679.755} C_VEL
LIN {X 0,Y 331.773,Z 621.554,A -85,B 0,C 180,E1 -14680.99,E2 -14680.99} C_VEL
LIN {X 0,Y 331.799,Z 622.678,A -85,B 0,C 180,E1 -14683.005,E2 -14683.005} C_VEL
LIN {X 0,Y 331.712,Z 622.752,A -85,B 0,C 180,E1 -14684.728,E2 -14684.728} C_VEL
LIN {X 0,Y 331.78,Z 622.341,A -85,B 0,C 180,E1 -14685.984,E2 -14685.984} C_VEL
LIN {X 0,Y 332.033,Z 621.018,A -85,B 0,C 180,E1 -14687.731,E2 -14687.731} C_VEL
LIN {X 0,Y 332.558,Z 617.371,A -85,B 0,C 180,E1 -14690.407,E2 -14690.407} C_VEL
LIN {X 0,Y 333.167,Z 613.47,A -85,B 0,C 180,E1 -14692.314,E2 -14692.314} C_VEL
LIN {X 0,Y 333.972,Z 608.337,A -85,B 0,C 180,E1 -14694.226,E2 -14694.226} C_VEL
LIN {X 0,Y 335.09,Z 601.808,A -85,B 0,C 180,E1 -14696.131,E2 -14696.131} C_VEL
LIN {X 0,Y 336.511,Z 593.517,A -85,B 0,C 180,E1 -14698.028,E2 -14698.028} C_VEL
LIN {X 0,Y 337.929,Z 584.967,A -85,B 0,C 180,E1 -14699.601,E2 -14699.601} C_VEL
LIN {X 0,Y 339.403,Z 575.607,A -85,B 0,C 180,E1 -14701.002,E2 -14701.002} C_VEL
LIN {X 0,Y 341.003,Z 564.479,A -85,B 0,C 180,E1 -14702.328,E2 -14702.328} C_VEL
LIN {X 0,Y 342.492,Z 552.196,A -85,B 0,C 180,E1 -14703.467,E2 -14703.467} C_VEL
LIN {X 0,Y 343.678,Z 540.236,A -85,B 0,C 180,E1 -14704.306,E2 -14704.306} C_VEL
LIN {X 0,Y 344.671,Z 527.378,A -85,B 0,C 180,E1 -14704.94,E2 -14704.94} C_VEL
LIN {X 0,Y 345.32,Z 514.141,A -85,B 0,C 180,E1 -14705.351,E2 -14705.351} C_VEL
LIN {X 0,Y 344.984,Z 508.345,A -85,B 0,C 180,E1 -14705.525,E2 -14705.525} C_VEL
LIN {X 0,Y 340.199,Z 489.726,A -85,B 0,C 180,E1 -14706.36,E2 -14706.36} C_VEL
LIN {X 0,Y 339.691,Z 483.921,A -85,B 0,C 180,E1 -14706.539,E2 -14706.539} C_VEL
LIN {X 0,Y 340.612,Z 444.959,A -85,B 0,C 180,E1 -14707.377,E2 -14707.377} C_VEL
LIN {X 0,Y 337.096,Z 428.848,A -85,B 0,C 180,E1 -14708.091,E2 -14708.091} C_VEL
LIN {X 0,Y 329.878,Z 412.335,A -85,B 0,C 180,E1 -14709.26,E2 -14709.26} C_VEL
LIN {X 0,Y 328.916,Z 407.94,A -85,B 0,C 180,E1 -14710.665,E2 -14710.665} C_VEL
LIN {X 0,Y 326.699,Z 398.383,A -85,B 0,C 180,E1 -14714.156,E2 -14714.156} C_VEL
LIN {X 0,Y 326.624,Z 398.29,A -85,B 0,C 180,E1 -14718.162,E2 -14718.162} C_VEL
LIN {X 0,Y 326.641,Z 398.287,A -85,B 0,C 180,E1 -14721.394,E2 -14721.394} C_VEL
LIN {X 0,Y 326.613,Z 398.288,A -85,B 0,C 180,E1 -14724.851,E2 -14724.851} C_VEL
LIN {X 0,Y 326.609,Z 398.303,A -85,B 0,C 180,E1 -14727.456,E2 -14727.456} C_VEL
LIN {X 0,Y 326.655,Z 398.275,A -85,B 0,C 180,E1 -14730.34,E2 -14730.34} C_VEL
LIN {X 0,Y 326.683,Z 398.289,A -85,B 0,C 180,E1 -14734.516,E2 -14734.516} C_VEL
LIN {X 0,Y 326.647,Z 398.29,A -85,B 0,C 180,E1 -14738.545,E2 -14738.545} C_VEL
LIN {X 0,Y 326.737,Z 398.279,A -85,B 0,C 180,E1 -14741.177,E2 -14741.177} C_VEL
LIN {X 0,Y 326.755,Z 398.274,A -85,B 0,C 180,E1 -14745.433,E2 -14745.433} C_VEL
LIN {X 0,Y 326.766,Z 398.276,A -85,B 0,C 180,E1 -14748.839,E2 -14748.839} C_VEL
LIN {X 0,Y 326.972,Z 398.258,A -85,B 0,C 180,E1 -14752.59,E2 -14752.59} C_VEL
LIN {X 0,Y 326.777,Z 398.273,A -85,B 0,C 180,E1 -14755.065,E2 -14755.065} C_VEL
LIN {X 0,Y 327.07,Z 398.24,A -85,B 0,C 180,E1 -14757.537,E2 -14757.537} C_VEL
LIN {X 0,Y 327.21,Z 398.219,A -85,B 0,C 180,E1 -14760,E2 -14760} C_VEL
LIN {X 0,Y 327.061,Z 398.244,A -85,B 0,C 180,E1 -14762.463,E2 -14762.463} C_VEL
LIN {X 0,Y 326.989,Z 398.253,A -85,B 0,C 180,E1 -14766.169,E2 -14766.169} C_VEL
LIN {X 0,Y 326.907,Z 398.255,A -85,B 0,C 180,E1 -14768.655,E2 -14768.655} C_VEL
LIN {X 0,Y 326.731,Z 398.283,A -85,B 0,C 180,E1 -14772.422,E2 -14772.422} C_VEL
LIN {X 0,Y 326.747,Z 398.281,A -85,B 0,C 180,E1 -14774.958,E2 -14774.958} C_VEL
LIN {X 0,Y 326.726,Z 398.279,A -85,B 0,C 180,E1 -14778.839,E2 -14778.839} C_VEL
LIN {X 0,Y 326.614,Z 398.292,A -85,B 0,C 180,E1 -14782.788,E2 -14782.788} C_VEL
LIN {X 0,Y 326.684,Z 398.289,A -85,B 0,C 180,E1 -14785.484,E2 -14785.484} C_VEL
LIN {X 0,Y 326.655,Z 398.293,A -85,B 0,C 180,E1 -14789.66,E2 -14789.66} C_VEL
LIN {X 0,Y 326.602,Z 398.297,A -85,B 0,C 180,E1 -14794.02,E2 -14794.02} C_VEL
LIN {X 0,Y 326.625,Z 398.294,A -85,B 0,C 180,E1 -14797.24,E2 -14797.24} C_VEL
LIN {X 0,Y 326.631,Z 398.288,A -85,B 0,C 180,E1 -14800.203,E2 -14800.203} C_VEL
LIN {X 0,Y 326.619,Z 398.299,A -85,B 0,C 180,E1 -14803.516,E2 -14803.516} C_VEL
LIN {X 0,Y 326.584,Z 398.293,A -85,B 0,C 180,E1 -14807.027,E2 -14807.027} C_VEL
LIN {X 0,Y 326.611,Z 398.293,A -85,B 0,C 180,E1 -14810.773,E2 -14810.773} C_VEL
LIN {X 0,Y 326.611,Z 398.299,A -85,B 0,C 180,E1 -14814.481,E2 -14814.481} C_VEL
LIN {X 0,Y 326.596,Z 398.363,A -85,B 0,C 180,E1 -14816.725,E2 -14816.725} C_VEL
LIN {X 0,Y 328.763,Z 407.12,A -85,B 0,C 180,E1 -14819.845,E2 -14819.845} C_VEL
LIN {X 0,Y 330.989,Z 417.12,A -85,B 0,C 180,E1 -14823.101,E2 -14823.101} C_VEL
LIN {X 0,Y 331.583,Z 420.24,A -85,B 0,C 180,E1 -14823.972,E2 -14823.972} C_VEL
LIN {X 0,Y 334.193,Z 426.957,A -85,B 0,C 180,E1 -14824.431,E2 -14824.431} C_VEL
LIN {X 0,Y 339.02,Z 449.227,A -85,B 0,C 180,E1 -14825.43,E2 -14825.43} C_VEL
LIN {X 0,Y 340.447,Z 457.974,A -85,B 0,C 180,E1 -14825.768,E2 -14825.768} C_VEL
LIN {X 0,Y 338.603,Z 528.294,A -85,B 0,C 180,E1 -14827.299,E2 -14827.299} C_VEL
LIN {X 0,Y 337.816,Z 541.239,A -85,B 0,C 180,E1 -14827.808,E2 -14827.808} C_VEL
LIN {X 0,Y 336.617,Z 553.244,A -85,B 0,C 180,E1 -14828.49,E2 -14828.49} C_VEL
LIN {X 0,Y 335.254,Z 565.383,A -85,B 0,C 180,E1 -14829.444,E2 -14829.444} C_VEL
LIN {X 0,Y 333.613,Z 576.886,A -85,B 0,C 180,E1 -14830.623,E2 -14830.623} C_VEL
LIN {X 0,Y 331.945,Z 587.258,A -85,B 0,C 180,E1 -14831.963,E2 -14831.963} C_VEL
LIN {X 0,Y 330.66,Z 595.226,A -85,B 0,C 180,E1 -14833.232,E2 -14833.232} C_VEL
LIN {X 0,Y 329.305,Z 603.598,A -85,B 0,C 180,E1 -14834.845,E2 -14834.845} C_VEL
LIN {X 0,Y 327.754,Z 611.305,A -85,B 0,C 180,E1 -14836.673,E2 -14836.673} C_VEL
LIN {X 0,Y 326.572,Z 618.394,A -85,B 0,C 180,E1 -14838.833,E2 -14838.833} C_VEL
LIN {X 0,Y 325.809,Z 623.138,A -85,B 0,C 180,E1 -14840.69,E2 -14840.69} C_VEL
LIN {X 0,Y 325.289,Z 626.786,A -85,B 0,C 180,E1 -14842.552,E2 -14842.552} C_VEL
LIN {X 0,Y 325.062,Z 628.968,A -85,B 0,C 180,E1 -14844.014,E2 -14844.014} C_VEL
LIN {X 0,Y 324.877,Z 631.163,A -85,B 0,C 180,E1 -14846.279,E2 -14846.279} C_VEL
LIN {X 0,Y 324.777,Z 632.077,A -85,B 0,C 180,E1 -14848.76,E2 -14848.76} C_VEL
LIN {X 0,Y 324.806,Z 631.937,A -85,B 0,C 180,E1 -14850,E2 -14850} C_VEL
LIN {X 0,Y 324.807,Z 630.424,A -85,B 0,C 180,E1 -14852.481,E2 -14852.481} C_VEL
LIN {X 0,Y 324.863,Z 629.076,A -85,B 0,C 180,E1 -14853.721,E2 -14853.721} C_VEL
LIN {X 0,Y 324.899,Z 626.003,A -85,B 0,C 180,E1 -14855.706,E2 -14855.706} C_VEL
LIN {X 0,Y 325.161,Z 622.304,A -85,B 0,C 180,E1 -14857.451,E2 -14857.451} C_VEL
LIN {X 0,Y 325.601,Z 617.252,A -85,B 0,C 180,E1 -14859.316,E2 -14859.316} C_VEL
LIN {X 0,Y 326.188,Z 610.881,A -85,B 0,C 180,E1 -14861.181,E2 -14861.181} C_VEL
LIN {X 0,Y 327.093,Z 602.885,A -85,B 0,C 180,E1 -14863.039,E2 -14863.039} C_VEL
LIN {X 0,Y 328.003,Z 594.721,A -85,B 0,C 180,E1 -14864.582,E2 -14864.582} C_VEL
LIN {X 0,Y 328.899,Z 586.052,A -85,B 0,C 180,E1 -14865.935,E2 -14865.935} C_VEL
LIN {X 0,Y 330.074,Z 574.913,A -85,B 0,C 180,E1 -14867.343,E2 -14867.343} C_VEL
LIN {X 0,Y 331.135,Z 564.242,A -85,B 0,C 180,E1 -14868.403,E2 -14868.403} C_VEL
LIN {X 0,Y 332.209,Z 551.369,A -85,B 0,C 180,E1 -14869.383,E2 -14869.383} C_VEL
LIN {X 0,Y 333.033,Z 538.378,A -85,B 0,C 180,E1 -14870.095,E2 -14870.095} C_VEL
LIN {X 0,Y 333.6,Z 525.528,A -85,B 0,C 180,E1 -14870.542,E2 -14870.542} C_VEL
LIN {X 0,Y 334.771,Z 454.651,A -85,B 0,C 180,E1 -14872.072,E2 -14872.072} C_VEL
LIN {X 0,Y 329.657,Z 420.645,A -85,B 0,C 180,E1 -14873.153,E2 -14873.153} C_VEL
LIN {X 0,Y 329.75,Z 418.588,A -85,B 0,C 180,E1 -14873.585,E2 -14873.585} C_VEL
LIN {X 0,Y 329.897,Z 415.016,A -85,B 0,C 180,E1 -14874.546,E2 -14874.546} C_VEL
LIN {X 0,Y 327.838,Z 403.745,A -85,B 0,C 180,E1 -14877.792,E2 -14877.792} C_VEL
LIN {X 0,Y 326.73,Z 398.343,A -85,B 0,C 180,E1 -14879.475,E2 -14879.475} C_VEL
LIN {X 0,Y 326.607,Z 398.298,A -85,B 0,C 180,E1 -14884.019,E2 -14884.019} C_VEL
LIN {X 0,Y 326.629,Z 398.299,A -85,B 0,C 180,E1 -14887.239,E2 -14887.239} C_VEL
LIN {X 0,Y 326.578,Z 398.304,A -85,B 0,C 180,E1 -14891.131,E2 -14891.131} C_VEL
LIN {X 0,Y 326.581,Z 398.298,A -85,B 0,C 180,E1 -14894.752,E2 -14894.752} C_VEL
LIN {X 0,Y 326.62,Z 398.295,A -85,B 0,C 180,E1 -14898.161,E2 -14898.161} C_VEL
LIN {X 0,Y 326.645,Z 398.299,A -85,B 0,C 180,E1 -14901.394,E2 -14901.394} C_VEL
LIN {X 0,Y 326.617,Z 398.296,A -85,B 0,C 180,E1 -14904.851,E2 -14904.851} C_VEL
LIN {X 0,Y 326.605,Z 398.305,A -85,B 0,C 180,E1 -14907.455,E2 -14907.455} C_VEL
LIN {X 0,Y 326.658,Z 398.29,A -85,B 0,C 180,E1 -14910.34,E2 -14910.34} C_VEL
LIN {X 0,Y 326.687,Z 398.288,A -85,B 0,C 180,E1 -14914.516,E2 -14914.516} C_VEL
LIN {X 0,Y 326.617,Z 398.295,A -85,B 0,C 180,E1 -14918.543,E2 -14918.543} C_VEL
LIN {X 0,Y 326.741,Z 398.281,A -85,B 0,C 180,E1 -14921.177,E2 -14921.177} C_VEL
LIN {X 0,Y 326.759,Z 398.284,A -85,B 0,C 180,E1 -14925.433,E2 -14925.433} C_VEL
LIN {X 0,Y 326.765,Z 398.277,A -85,B 0,C 180,E1 -14928.839,E2 -14928.839} C_VEL
LIN {X 0,Y 326.954,Z 398.254,A -85,B 0,C 180,E1 -14932.59,E2 -14932.59} C_VEL
LIN {X 0,Y 326.773,Z 398.281,A -85,B 0,C 180,E1 -14935.065,E2 -14935.065} C_VEL
LIN {X 0,Y 327.043,Z 398.245,A -85,B 0,C 180,E1 -14937.537,E2 -14937.537} C_VEL
LIN {X 0,Y 327.193,Z 398.22,A -85,B 0,C 180,E1 -14940,E2 -14940} C_VEL
LIN {X 0,Y 327.043,Z 398.24,A -85,B 0,C 180,E1 -14942.463,E2 -14942.463} C_VEL
LIN {X 0,Y 326.955,Z 398.254,A -85,B 0,C 180,E1 -14946.652,E2 -14946.652} C_VEL
LIN {X 0,Y 326.801,Z 398.272,A -85,B 0,C 180,E1 -14949.907,E2 -14949.907} C_VEL
LIN {X 0,Y 326.754,Z 398.278,A -85,B 0,C 180,E1 -14953.686,E2 -14953.686} C_VEL
LIN {X 0,Y 326.695,Z 398.29,A -85,B 0,C 180,E1 -14957.528,E2 -14957.528} C_VEL
LIN {X 0,Y 326.661,Z 398.291,A -85,B 0,C 180,E1 -14960.135,E2 -14960.135} C_VEL
LIN {X 0,Y 326.648,Z 398.288,A -85,B 0,C 180,E1 -14964.129,E2 -14964.129} C_VEL
LIN {X 0,Y 326.682,Z 398.29,A -85,B 0,C 180,E1 -14966.858,E2 -14966.858} C_VEL
LIN {X 0,Y 326.636,Z 398.295,A -85,B 0,C 180,E1 -14970.611,E2 -14970.611} C_VEL
LIN {X 0,Y 326.604,Z 398.294,A -85,B 0,C 180,E1 -14974.02,E2 -14974.02} C_VEL
LIN {X 0,Y 326.625,Z 398.301,A -85,B 0,C 180,E1 -14977.239,E2 -14977.239} C_VEL
LIN {X 0,Y 326.575,Z 398.303,A -85,B 0,C 180,E1 -14981.132,E2 -14981.132} C_VEL
LIN {X 0,Y 326.558,Z 398.306,A -85,B 0,C 180,E1 -14984.749,E2 -14984.749} C_VEL
LIN {X 0,Y 326.597,Z 398.298,A -85,B 0,C 180,E1 -14988.158,E2 -14988.158} C_VEL
LIN {X 0,Y 326.642,Z 398.297,A -85,B 0,C 180,E1 -14991.395,E2 -14991.395} C_VEL
LIN {X 0,Y 326.619,Z 398.3,A -85,B 0,C 180,E1 -14994.851,E2 -14994.851} C_VEL
LIN {X 0,Y 326.607,Z 398.294,A -85,B 0,C 180,E1 -14997.456,E2 -14997.456} C_VEL
LIN {X 0,Y 326.66,Z 398.291,A -85,B 0,C 180,E1 -15000.341,E2 -15000.341} C_VEL
LIN {X 0,Y 326.69,Z 398.287,A -85,B 0,C 180,E1 -15004.517,E2 -15004.517} C_VEL
LIN {X 0,Y 326.649,Z 398.296,A -85,B 0,C 180,E1 -15008.546,E2 -15008.546} C_VEL
LIN {X 0,Y 326.745,Z 398.276,A -85,B 0,C 180,E1 -15011.178,E2 -15011.178} C_VEL
LIN {X 0,Y 326.764,Z 398.284,A -85,B 0,C 180,E1 -15015.433,E2 -15015.433} C_VEL
LIN {X 0,Y 326.813,Z 398.447,A -85,B 0,C 180,E1 -15015.757,E2 -15015.757} C_VEL
LIN {X 0,Y 328.716,Z 408.574,A -85,B 0,C 180,E1 -15018.906,E2 -15018.906} C_VEL
LIN {X 0,Y 329.337,Z 412.03,A -85,B 0,C 180,E1 -15019.864,E2 -15019.864} C_VEL
LIN {X 0,Y 330.72,Z 417.659,A -85,B 0,C 180,E1 -15020.117,E2 -15020.117} C_VEL
LIN {X 0,Y 333.823,Z 435.814,A -85,B 0,C 180,E1 -15020.705,E2 -15020.705} C_VEL
LIN {X 0,Y 335.035,Z 443.545,A -85,B 0,C 180,E1 -15020.948,E2 -15020.948} C_VEL
LIN {X 0,Y 333.545,Z 518.879,A -85,B 0,C 180,E1 -15022.574,E2 -15022.574} C_VEL
LIN {X 0,Y 333.013,Z 531.865,A -85,B 0,C 180,E1 -15023.084,E2 -15023.084} C_VEL
LIN {X 0,Y 332.248,Z 544.446,A -85,B 0,C 180,E1 -15023.818,E2 -15023.818} C_VEL
LIN {X 0,Y 331.308,Z 555.41,A -85,B 0,C 180,E1 -15024.675,E2 -15024.675} C_VEL
LIN {X 0,Y 330.1,Z 567.26,A -85,B 0,C 180,E1 -15025.879,E2 -15025.879} C_VEL
LIN {X 0,Y 328.933,Z 577.841,A -85,B 0,C 180,E1 -15027.244,E2 -15027.244} C_VEL
LIN {X 0,Y 327.898,Z 587.368,A -85,B 0,C 180,E1 -15028.772,E2 -15028.772} C_VEL
LIN {X 0,Y 327.052,Z 595.168,A -85,B 0,C 180,E1 -15030.307,E2 -15030.307} C_VEL
LIN {X 0,Y 326.221,Z 602.795,A -85,B 0,C 180,E1 -15032.16,E2 -15032.16} C_VEL
LIN {X 0,Y 325.477,Z 609.848,A -85,B 0,C 180,E1 -15034.334,E2 -15034.334} C_VEL
LIN {X 0,Y 325.231,Z 614.658,A -85,B 0,C 180,E1 -15036.265,E2 -15036.265} C_VEL
LIN {X 0,Y 324.944,Z 618.088,A -85,B 0,C 180,E1 -15038.081,E2 -15038.081} C_VEL
LIN {X 0,Y 324.708,Z 620.642,A -85,B 0,C 180,E1 -15039.971,E2 -15039.971} C_VEL
LIN {X 0,Y 324.691,Z 621.82,A -85,B 0,C 180,E1 -15041.233,E2 -15041.233} C_VEL
LIN {X 0,Y 324.713,Z 622.784,A -85,B 0,C 180,E1 -15043.102,E2 -15043.102} C_VEL
LIN {X 0,Y 324.627,Z 622.828,A -85,B 0,C 180,E1 -15045.057,E2 -15045.057} C_VEL
LIN {X 0,Y 324.725,Z 622.32,A -85,B 0,C 180,E1 -15046.341,E2 -15046.341} C_VEL
LIN {X 0,Y 324.978,Z 621.127,A -85,B 0,C 180,E1 -15047.909,E2 -15047.909} C_VEL
LIN {X 0,Y 325.407,Z 618.214,A -85,B 0,C 180,E1 -15050.215,E2 -15050.215} C_VEL
LIN {X 0,Y 325.969,Z 614.894,A -85,B 0,C 180,E1 -15052.014,E2 -15052.014} C_VEL
LIN {X 0,Y 326.818,Z 609.705,A -85,B 0,C 180,E1 -15054.115,E2 -15054.115} C_VEL
LIN {X 0,Y 328.017,Z 603.122,A -85,B 0,C 180,E1 -15056.16,E2 -15056.16} C_VEL
LIN {X 0,Y 329.394,Z 595.665,A -85,B 0,C 180,E1 -15057.994,E2 -15057.994} C_VEL
LIN {X 0,Y 330.972,Z 586.759,A -85,B 0,C 180,E1 -15059.74,E2 -15059.74} C_VEL
LIN {X 0,Y 332.504,Z 577.613,A -85,B 0,C 180,E1 -15061.187,E2 -15061.187} C_VEL
LIN {X 0,Y 334.063,Z 567.514,A -85,B 0,C 180,E1 -15062.48,E2 -15062.48} C_VEL
LIN {X 0,Y 335.66,Z 555.467,A -85,B 0,C 180,E1 -15063.699,E2 -15063.699} C_VEL
LIN {X 0,Y 336.987,Z 543.259,A -85,B 0,C 180,E1 -15064.631,E2 -15064.631} C_VEL
LIN {X 0,Y 338.129,Z 530.027,A -85,B 0,C 180,E1 -15065.36,E2 -15065.36} C_VEL
LIN {X 0,Y 338.846,Z 517.393,A -85,B 0,C 180,E1 -15065.806,E2 -15065.806} C_VEL
LIN {X 0,Y 339.691,Z 483.921,A -85,B 0,C 180,E1 -15066.539,E2 -15066.539} C_VEL
LIN {X 0,Y 339.245,Z 478.123,A -85,B 0,C 180,E1 -15066.715,E2 -15066.715} C_VEL
LIN {X 0,Y 334.773,Z 459.467,A -85,B 0,C 180,E1 -15067.569,E2 -15067.569} C_VEL
LIN {X 0,Y 334.259,Z 453.674,A -85,B 0,C 180,E1 -15067.759,E2 -15067.759} C_VEL
LIN {X 0,Y 334.279,Z 445.589,A -85,B 0,C 180,E1 -15067.954,E2 -15067.954} C_VEL
LIN {X 0,Y 331.236,Z 431.686,A -85,B 0,C 180,E1 -15068.595,E2 -15068.595} C_VEL
LIN {X 0,Y 324.094,Z 415.539,A -85,B 0,C 180,E1 -15069.744,E2 -15069.744} C_VEL
LIN {X 0,Y 322.655,Z 412.22,A -85,B 0,C 180,E1 -15070.055,E2 -15070.055} C_VEL
LIN {X 0,Y 320.739,Z 403.825,A -85,B 0,C 180,E1 -15073.018,E2 -15073.018} C_VEL
LIN {X 0,Y 319.638,Z 399.19,A -85,B 0,C 180,E1 -15074.864,E2 -15074.864} C_VEL
LIN {X 0,Y 319.578,Z 399.171,A -85,B 0,C 180,E1 -15078.72,E2 -15078.72} C_VEL
LIN {X 0,Y 319.593,Z 399.171,A -85,B 0,C 180,E1 -15082.339,E2 -15082.339} C_VEL
LIN {X 0,Y 319.554,Z 399.165,A -85,B 0,C 180,E1 -15085.123,E2 -15085.123} C_VEL
LIN {X 0,Y 319.568,Z 399.166,A -85,B 0,C 180,E1 -15089.056,E2 -15089.056} C_VEL
LIN {X 0,Y 319.602,Z 399.173,A -85,B 0,C 180,E1 -15092.498,E2 -15092.498} C_VEL
LIN {X 0,Y 319.599,Z 399.173,A -85,B 0,C 180,E1 -15095.304,E2 -15095.304} C_VEL
LIN {X 0,Y 319.617,Z 399.173,A -85,B 0,C 180,E1 -15099.401,E2 -15099.401} C_VEL
LIN {X 0,Y 319.651,Z 399.161,A -85,B 0,C 180,E1 -15102.073,E2 -15102.073} C_VEL
LIN {X 0,Y 319.725,Z 399.151,A -85,B 0,C 180,E1 -15106.008,E2 -15106.008} C_VEL
LIN {X 0,Y 319.752,Z 399.144,A -85,B 0,C 180,E1 -15109.873,E2 -15109.873} C_VEL
LIN {X 0,Y 319.926,Z 399.134,A -85,B 0,C 180,E1 -15112.426,E2 -15112.426} C_VEL
LIN {X 0,Y 319.746,Z 399.148,A -85,B 0,C 180,E1 -15114.956,E2 -15114.956} C_VEL
LIN {X 0,Y 320.01,Z 399.12,A -85,B 0,C 180,E1 -15117.483,E2 -15117.483} C_VEL
LIN {X 0,Y 320.162,Z 399.097,A -85,B 0,C 180,E1 -15120,E2 -15120} C_VEL
LIN {X 0,Y 320.001,Z 399.122,A -85,B 0,C 180,E1 -15122.518,E2 -15122.518} C_VEL
LIN {X 0,Y 319.945,Z 399.131,A -85,B 0,C 180,E1 -15126.306,E2 -15126.306} C_VEL
LIN {X 0,Y 319.836,Z 399.135,A -85,B 0,C 180,E1 -15128.848,E2 -15128.848} C_VEL
LIN {X 0,Y 319.678,Z 399.157,A -85,B 0,C 180,E1 -15132.7,E2 -15132.7} C_VEL
LIN {X 0,Y 319.692,Z 399.162,A -85,B 0,C 180,E1 -15135.296,E2 -15135.296} C_VEL
LIN {X 0,Y 319.668,Z 399.161,A -85,B 0,C 180,E1 -15139.256,E2 -15139.256} C_VEL
LIN {X 0,Y 319.564,Z 399.172,A -85,B 0,C 180,E1 -15143.32,E2 -15143.32} C_VEL
LIN {X 0,Y 319.629,Z 399.166,A -85,B 0,C 180,E1 -15146.089,E2 -15146.089} C_VEL
LIN {X 0,Y 319.584,Z 399.176,A -85,B 0,C 180,E1 -15148.934,E2 -15148.934} C_VEL
LIN {X 0,Y 319.526,Z 399.181,A -85,B 0,C 180,E1 -15151.863,E2 -15151.863} C_VEL
LIN {X 0,Y 319.575,Z 399.177,A -85,B 0,C 180,E1 -15155.544,E2 -15155.544} C_VEL
LIN {X 0,Y 319.595,Z 399.171,A -85,B 0,C 180,E1 -15158.005,E2 -15158.005} C_VEL
LIN {X 0,Y 319.592,Z 399.153,A -85,B 0,C 180,E1 -15161.612,E2 -15161.612} C_VEL
LIN {X 0,Y 319.54,Z 399.174,A -85,B 0,C 180,E1 -15165.268,E2 -15165.268} C_VEL
LIN {X 0,Y 319.53,Z 399.182,A -85,B 0,C 180,E1 -15168.713,E2 -15168.713} C_VEL
LIN {X 0,Y 319.575,Z 399.176,A -85,B 0,C 180,E1 -15172.345,E2 -15172.345} C_VEL
LIN {X 0,Y 319.565,Z 399.248,A -85,B 0,C 180,E1 -15176.08,E2 -15176.08} C_VEL
LIN {X 0,Y 321.654,Z 407.624,A -85,B 0,C 180,E1 -15179.164,E2 -15179.164} C_VEL
LIN {X 0,Y 323.671,Z 416.517,A -85,B 0,C 180,E1 -15182.172,E2 -15182.172} C_VEL
LIN {X 0,Y 324.381,Z 420.018,A -85,B 0,C 180,E1 -15183.218,E2 -15183.218} C_VEL
LIN {X 0,Y 328.235,Z 429.226,A -85,B 0,C 180,E1 -15183.89,E2 -15183.89} C_VEL
LIN {X 0,Y 332.91,Z 450.943,A -85,B 0,C 180,E1 -15184.897,E2 -15184.897} C_VEL
LIN {X 0,Y 334.184,Z 458.968,A -85,B 0,C 180,E1 -15185.214,E2 -15185.214} C_VEL
LIN {X 0,Y 332.271,Z 528.503,A -85,B 0,C 180,E1 -15186.759,E2 -15186.759} C_VEL
LIN {X 0,Y 331.328,Z 542.114,A -85,B 0,C 180,E1 -15187.308,E2 -15187.308} C_VEL
LIN {X 0,Y 330.083,Z 554.399,A -85,B 0,C 180,E1 -15188.042,E2 -15188.042} C_VEL
LIN {X 0,Y 328.675,Z 566.175,A -85,B 0,C 180,E1 -15189.013,E2 -15189.013} C_VEL
LIN {X 0,Y 326.957,Z 577.518,A -85,B 0,C 180,E1 -15190.212,E2 -15190.212} C_VEL
LIN {X 0,Y 325.216,Z 587.764,A -85,B 0,C 180,E1 -15191.577,E2 -15191.577} C_VEL
LIN {X 0,Y 323.819,Z 596.031,A -85,B 0,C 180,E1 -15192.941,E2 -15192.941} C_VEL
LIN {X 0,Y 322.459,Z 603.904,A -85,B 0,C 180,E1 -15194.515,E2 -15194.515} C_VEL
LIN {X 0,Y 320.84,Z 611.509,A -85,B 0,C 180,E1 -15196.381,E2 -15196.381} C_VEL
LIN {X 0,Y 319.609,Z 618.536,A -85,B 0,C 180,E1 -15198.586,E2 -15198.586} C_VEL
LIN {X 0,Y 318.805,Z 623.228,A -85,B 0,C 180,E1 -15200.484,E2 -15200.484} C_VEL
LIN {X 0,Y 318.228,Z 626.828,A -85,B 0,C 180,E1 -15202.386,E2 -15202.386} C_VEL
LIN {X 0,Y 317.979,Z 629.148,A -85,B 0,C 180,E1 -15204.041,E2 -15204.041} C_VEL
LIN {X 0,Y 317.79,Z 631.116,A -85,B 0,C 180,E1 -15206.196,E2 -15206.196} C_VEL
LIN {X 0,Y 317.731,Z 631.743,A -85,B 0,C 180,E1 -15207.465,E2 -15207.465} C_VEL
LIN {X 0,Y 317.691,Z 631.986,A -85,B 0,C 180,E1 -15208.733,E2 -15208.733} C_VEL
LIN {X 0,Y 317.717,Z 631.804,A -85,B 0,C 180,E1 -15210,E2 -15210} C_VEL
LIN {X 0,Y 317.73,Z 630.248,A -85,B 0,C 180,E1 -15212.536,E2 -15212.536} C_VEL
LIN {X 0,Y 317.774,Z 628.877,A -85,B 0,C 180,E1 -15213.805,E2 -15213.805} C_VEL
LIN {X 0,Y 317.8,Z 626.083,A -85,B 0,C 180,E1 -15215.641,E2 -15215.641} C_VEL
LIN {X 0,Y 318.09,Z 622.01,A -85,B 0,C 180,E1 -15217.618,E2 -15217.618} C_VEL
LIN {X 0,Y 318.65,Z 615.908,A -85,B 0,C 180,E1 -15219.842,E2 -15219.842} C_VEL
LIN {X 0,Y 319.309,Z 609.206,A -85,B 0,C 180,E1 -15221.747,E2 -15221.747} C_VEL
LIN {X 0,Y 320.352,Z 600.882,A -85,B 0,C 180,E1 -15223.641,E2 -15223.641} C_VEL
LIN {X 0,Y 321.368,Z 592.32,A -85,B 0,C 180,E1 -15225.214,E2 -15225.214} C_VEL
LIN {X 0,Y 322.436,Z 581.7,A -85,B 0,C 180,E1 -15226.786,E2 -15226.786} C_VEL
LIN {X 0,Y 323.53,Z 571.177,A -85,B 0,C 180,E1 -15228.032,E2 -15228.032} C_VEL
LIN {X 0,Y 324.679,Z 559.588,A -85,B 0,C 180,E1 -15229.111,E2 -15229.111} C_VEL
LIN {X 0,Y 325.668,Z 547.538,A -85,B 0,C 180,E1 -15229.952,E2 -15229.952} C_VEL
LIN {X 0,Y 326.449,Z 534.474,A -85,B 0,C 180,E1 -15230.601,E2 -15230.601} C_VEL
LIN {X 0,Y 326.911,Z 522.171,A -85,B 0,C 180,E1 -15230.982,E2 -15230.982} C_VEL
LIN {X 0,Y 328.044,Z 455.469,A -85,B 0,C 180,E1 -15232.439,E2 -15232.439} C_VEL
LIN {X 0,Y 322.786,Z 420.267,A -85,B 0,C 180,E1 -15233.601,E2 -15233.601} C_VEL
LIN {X 0,Y 322.991,Z 417.012,A -85,B 0,C 180,E1 -15234.42,E2 -15234.42} C_VEL
LIN {X 0,Y 321.029,Z 405.761,A -85,B 0,C 180,E1 -15237.722,E2 -15237.722} C_VEL
LIN {X 0,Y 319.677,Z 399.205,A -85,B 0,C 180,E1 -15239.805,E2 -15239.805} C_VEL
LIN {X 0,Y 319.577,Z 399.179,A -85,B 0,C 180,E1 -15243.352,E2 -15243.352} C_VEL
LIN {X 0,Y 319.56,Z 399.177,A -85,B 0,C 180,E1 -15246.427,E2 -15246.427} C_VEL
LIN {X 0,Y 319.558,Z 399.178,A -85,B 0,C 180,E1 -15249.668,E2 -15249.668} C_VEL
LIN {X 0,Y 319.563,Z 399.177,A -85,B 0,C 180,E1 -15253.468,E2 -15253.468} C_VEL
LIN {X 0,Y 319.601,Z 399.163,A -85,B 0,C 180,E1 -15257.024,E2 -15257.024} C_VEL
LIN {X 0,Y 319.584,Z 399.174,A -85,B 0,C 180,E1 -15260.376,E2 -15260.376} C_VEL
LIN {X 0,Y 319.557,Z 399.178,A -85,B 0,C 180,E1 -15263.572,E2 -15263.572} C_VEL
LIN {X 0,Y 319.575,Z 399.175,A -85,B 0,C 180,E1 -15266.686,E2 -15266.686} C_VEL
LIN {X 0,Y 319.588,Z 399.174,A -85,B 0,C 180,E1 -15269.616,E2 -15269.616} C_VEL
LIN {X 0,Y 319.605,Z 399.168,A -85,B 0,C 180,E1 -15272.498,E2 -15272.498} C_VEL
LIN {X 0,Y 319.6,Z 399.176,A -85,B 0,C 180,E1 -15275.303,E2 -15275.303} C_VEL
LIN {X 0,Y 319.6,Z 399.17,A -85,B 0,C 180,E1 -15279.4,E2 -15279.4} C_VEL
LIN {X 0,Y 319.654,Z 399.164,A -85,B 0,C 180,E1 -15282.073,E2 -15282.073} C_VEL
LIN {X 0,Y 319.728,Z 399.155,A -85,B 0,C 180,E1 -15286.007,E2 -15286.007} C_VEL
LIN {X 0,Y 319.748,Z 399.148,A -85,B 0,C 180,E1 -15289.872,E2 -15289.872} C_VEL
LIN {X 0,Y 319.908,Z 399.131,A -85,B 0,C 180,E1 -15292.426,E2 -15292.426} C_VEL
LIN {X 0,Y 319.742,Z 399.156,A -85,B 0,C 180,E1 -15294.956,E2 -15294.956} C_VEL
LIN {X 0,Y 319.987,Z 399.124,A -85,B 0,C 180,E1 -15297.482,E2 -15297.482} C_VEL
LIN {X 0,Y 320.145,Z 399.097,A -85,B 0,C 180,E1 -15300,E2 -15300} C_VEL
LIN {X 0,Y 319.987,Z 399.118,A -85,B 0,C 180,E1 -15302.518,E2 -15302.518} C_VEL
LIN {X 0,Y 319.916,Z 399.13,A -85,B 0,C 180,E1 -15306.64,E2 -15306.64} C_VEL
LIN {X 0,Y 319.748,Z 399.149,A -85,B 0,C 180,E1 -15310.127,E2 -15310.127} C_VEL
LIN {X 0,Y 319.727,Z 399.152,A -85,B 0,C 180,E1 -15314.724,E2 -15314.724} C_VEL
LIN {X 0,Y 319.685,Z 399.165,A -85,B 0,C 180,E1 -15319.038,E2 -15319.038} C_VEL
LIN {X 0,Y 319.566,Z 399.172,A -85,B 0,C 180,E1 -15323.32,E2 -15323.32} C_VEL
LIN {X 0,Y 319.631,Z 399.165,A -85,B 0,C 180,E1 -15326.088,E2 -15326.088} C_VEL
LIN {X 0,Y 319.587,Z 399.176,A -85,B 0,C 180,E1 -15328.934,E2 -15328.934} C_VEL
LIN {X 0,Y 319.529,Z 399.177,A -85,B 0,C 180,E1 -15331.862,E2 -15331.862} C_VEL
LIN {X 0,Y 319.577,Z 399.175,A -85,B 0,C 180,E1 -15335.543,E2 -15335.543} C_VEL
LIN {X 0,Y 319.556,Z 399.176,A -85,B 0,C 180,E1 -15339.669,E2 -15339.669} C_VEL
LIN {X 0,Y 319.555,Z 399.178,A -85,B 0,C 180,E1 -15343.468,E2 -15343.468} C_VEL
LIN {X 0,Y 319.58,Z 399.179,A -85,B 0,C 180,E1 -15347.022,E2 -15347.022} C_VEL
LIN {X 0,Y 319.581,Z 399.173,A -85,B 0,C 180,E1 -15350.376,E2 -15350.376} C_VEL
LIN {X 0,Y 319.559,Z 399.177,A -85,B 0,C 180,E1 -15353.573,E2 -15353.573} C_VEL
LIN {X 0,Y 319.576,Z 399.17,A -85,B 0,C 180,E1 -15356.687,E2 -15356.687} C_VEL
LIN {X 0,Y 319.591,Z 399.172,A -85,B 0,C 180,E1 -15359.617,E2 -15359.617} C_VEL
LIN {X 0,Y 319.608,Z 399.172,A -85,B 0,C 180,E1 -15362.498,E2 -15362.498} C_VEL
LIN {X 0,Y 319.605,Z 399.168,A -85,B 0,C 180,E1 -15365.304,E2 -15365.304} C_VEL
LIN {X 0,Y 319.598,Z 399.172,A -85,B 0,C 180,E1 -15368.048,E2 -15368.048} C_VEL
LIN {X 0,Y 319.69,Z 399.154,A -85,B 0,C 180,E1 -15370.962,E2 -15370.962} C_VEL
LIN {X 0,Y 319.75,Z 399.236,A -85,B 0,C 180,E1 -15375.403,E2 -15375.403} C_VEL
LIN {X 0,Y 321.663,Z 409.398,A -85,B 0,C 180,E1 -15378.659,E2 -15378.659} C_VEL
LIN {X 0,Y 322.163,Z 412.175,A -85,B 0,C 180,E1 -15379.427,E2 -15379.427} C_VEL
LIN {X 0,Y 324.026,Z 418.562,A -85,B 0,C 180,E1 -15379.726,E2 -15379.726} C_VEL
LIN {X 0,Y 327.314,Z 437.874,A -85,B 0,C 180,E1 -15380.37,E2 -15380.37} C_VEL
LIN {X 0,Y 328.301,Z 444.553,A -85,B 0,C 180,E1 -15380.581,E2 -15380.581} C_VEL
LIN {X 0,Y 326.765,Z 518.881,A -85,B 0,C 180,E1 -15382.215,E2 -15382.215} C_VEL
LIN {X 0,Y 326.207,Z 532.015,A -85,B 0,C 180,E1 -15382.74,E2 -15382.74} C_VEL
LIN {X 0,Y 325.443,Z 544.314,A -85,B 0,C 180,E1 -15383.471,E2 -15383.471} C_VEL
LIN {X 0,Y 324.404,Z 556.011,A -85,B 0,C 180,E1 -15384.405,E2 -15384.405} C_VEL
LIN {X 0,Y 323.158,Z 567.739,A -85,B 0,C 180,E1 -15385.634,E2 -15385.634} C_VEL
LIN {X 0,Y 321.956,Z 578.255,A -85,B 0,C 180,E1 -15387.028,E2 -15387.028} C_VEL
LIN {X 0,Y 320.965,Z 586.844,A -85,B 0,C 180,E1 -15388.431,E2 -15388.431} C_VEL
LIN {X 0,Y 320.108,Z 594.753,A -85,B 0,C 180,E1 -15390,E2 -15390} C_VEL
LIN {X 0,Y 319.198,Z 602.503,A -85,B 0,C 180,E1 -15391.892,E2 -15391.892} C_VEL
LIN {X 0,Y 318.494,Z 608.719,A -85,B 0,C 180,E1 -15393.795,E2 -15393.795} C_VEL
LIN {X 0,Y 318.162,Z 614.03,A -85,B 0,C 180,E1 -15395.875,E2 -15395.875} C_VEL
LIN {X 0,Y 317.918,Z 617.456,A -85,B 0,C 180,E1 -15397.622,E2 -15397.622} C_VEL
LIN {X 0,Y 317.723,Z 619.429,A -85,B 0,C 180,E1 -15398.907,E2 -15398.907} C_VEL
LIN {X 0,Y 317.594,Z 620.975,A -85,B 0,C 180,E1 -15400.196,E2 -15400.196} C_VEL
LIN {X 0,Y 317.596,Z 622.053,A -85,B 0,C 180,E1 -15401.487,E2 -15401.487} C_VEL
LIN {X 0,Y 317.616,Z 622.886,A -85,B 0,C 180,E1 -15403.194,E2 -15403.194} C_VEL
LIN {X 0,Y 317.553,Z 622.876,A -85,B 0,C 180,E1 -15405.401,E2 -15405.401} C_VEL
LIN {X 0,Y 317.692,Z 622.289,A -85,B 0,C 180,E1 -15406.713,E2 -15406.713} C_VEL
LIN {X 0,Y 317.927,Z 621.236,A -85,B 0,C 180,E1 -15408.094,E2 -15408.094} C_VEL
LIN {X 0,Y 318.113,Z 619.877,A -85,B 0,C 180,E1 -15409.353,E2 -15409.353} C_VEL
LIN {X 0,Y 318.644,Z 616.849,A -85,B 0,C 180,E1 -15411.341,E2 -15411.341} C_VEL
LIN {X 0,Y 319.367,Z 612.685,A -85,B 0,C 180,E1 -15413.334,E2 -15413.334} C_VEL
LIN {X 0,Y 320.6,Z 606.199,A -85,B 0,C 180,E1 -15415.654,E2 -15415.654} C_VEL
LIN {X 0,Y 321.981,Z 599.066,A -85,B 0,C 180,E1 -15417.634,E2 -15417.634} C_VEL
LIN {X 0,Y 323.365,Z 591.925,A -85,B 0,C 180,E1 -15419.226,E2 -15419.226} C_VEL
LIN {X 0,Y 325.008,Z 582.688,A -85,B 0,C 180,E1 -15420.901,E2 -15420.901} C_VEL
LIN {X 0,Y 326.756,Z 572.73,A -85,B 0,C 180,E1 -15422.344,E2 -15422.344} C_VEL
LIN {X 0,Y 328.39,Z 561.786,A -85,B 0,C 180,E1 -15423.619,E2 -15423.619} C_VEL
LIN {X 0,Y 329.836,Z 550.38,A -85,B 0,C 180,E1 -15424.655,E2 -15424.655} C_VEL
LIN {X 0,Y 331.14,Z 537.614,A -85,B 0,C 180,E1 -15425.52,E2 -15425.52} C_VEL
LIN {X 0,Y 332.157,Z 524.384,A -85,B 0,C 180,E1 -15426.141,E2 -15426.141} C_VEL
LIN {X 0,Y 332.777,Z 509.393,A -85,B 0,C 180,E1 -15426.548,E2 -15426.548} C_VEL
LIN {X 0,Y 334.259,Z 453.674,A -85,B 0,C 180,E1 -15427.759,E2 -15427.759} C_VEL
LIN {X 0,Y 333.87,Z 449.844,A -85,B 0,C 180,E1 -15427.889,E2 -15427.889} C_VEL
LIN {X 0,Y 332.149,Z 444.449,A -85,B 0,C 180,E1 -15428.189,E2 -15428.189} C_VEL
LIN {X 0,Y 329.589,Z 439.498,A -85,B 0,C 180,E1 -15428.566,E2 -15428.566} C_VEL
LIN {X 0,Y 325.57,Z 433.068,A -85,B 0,C 180,E1 -15429.138,E2 -15429.138} C_VEL
LIN {X 0,Y 321.952,Z 426.371,A -85,B 0,C 180,E1 -15429.693,E2 -15429.693} C_VEL
LIN {X 0,Y 316.219,Z 414.318,A -85,B 0,C 180,E1 -15430.644,E2 -15430.644} C_VEL
LIN {X 0,Y 315.424,Z 412.184,A -85,B 0,C 180,E1 -15430.89,E2 -15430.89} C_VEL
LIN {X 0,Y 313.395,Z 403.38,A -85,B 0,C 180,E1 -15434.142,E2 -15434.142} C_VEL
LIN {X 0,Y 312.586,Z 400.071,A -85,B 0,C 180,E1 -15435.533,E2 -15435.533} C_VEL
LIN {X 0,Y 312.523,Z 400.056,A -85,B 0,C 180,E1 -15439.296,E2 -15439.296} C_VEL
LIN {X 0,Y 312.547,Z 400.051,A -85,B 0,C 180,E1 -15442.618,E2 -15442.618} C_VEL
LIN {X 0,Y 312.514,Z 400.047,A -85,B 0,C 180,E1 -15446.31,E2 -15446.31} C_VEL
LIN {X 0,Y 312.54,Z 400.032,A -85,B 0,C 180,E1 -15450.35,E2 -15450.35} C_VEL
LIN {X 0,Y 312.596,Z 400.045,A -85,B 0,C 180,E1 -15454.064,E2 -15454.064} C_VEL
LIN {X 0,Y 312.581,Z 400.042,A -85,B 0,C 180,E1 -15457.529,E2 -15457.529} C_VEL
LIN {X 0,Y 312.632,Z 400.034,A -85,B 0,C 180,E1 -15461.656,E2 -15461.656} C_VEL
LIN {X 0,Y 312.687,Z 400.026,A -85,B 0,C 180,E1 -15465.686,E2 -15465.686} C_VEL
LIN {X 0,Y 312.696,Z 400.023,A -85,B 0,C 180,E1 -15469.642,E2 -15469.642} C_VEL
LIN {X 0,Y 312.864,Z 400.013,A -85,B 0,C 180,E1 -15472.254,E2 -15472.254} C_VEL
LIN {X 0,Y 312.715,Z 400.023,A -85,B 0,C 180,E1 -15474.842,E2 -15474.842} C_VEL
LIN {X 0,Y 312.954,Z 399.999,A -85,B 0,C 180,E1 -15477.426,E2 -15477.426} C_VEL
LIN {X 0,Y 313.113,Z 399.975,A -85,B 0,C 180,E1 -15480,E2 -15480} C_VEL
LIN {X 0,Y 312.945,Z 400,A -85,B 0,C 180,E1 -15482.574,E2 -15482.574} C_VEL
LIN {X 0,Y 312.903,Z 400.009,A -85,B 0,C 180,E1 -15486.448,E2 -15486.448} C_VEL
LIN {X 0,Y 312.781,Z 400.014,A -85,B 0,C 180,E1 -15489.05,E2 -15489.05} C_VEL
LIN {X 0,Y 312.63,Z 400.032,A -85,B 0,C 180,E1 -15492.991,E2 -15492.991} C_VEL
LIN {X 0,Y 312.631,Z 400.041,A -85,B 0,C 180,E1 -15495.65,E2 -15495.65} C_VEL
LIN {X 0,Y 312.624,Z 400.038,A -85,B 0,C 180,E1 -15499.237,E2 -15499.237} C_VEL
LIN {X 0,Y 312.539,Z 400.045,A -85,B 0,C 180,E1 -15502.79,E2 -15502.79} C_VEL
LIN {X 0,Y 312.597,Z 400.043,A -85,B 0,C 180,E1 -15505.936,E2 -15505.936} C_VEL
LIN {X 0,Y 312.539,Z 400.051,A -85,B 0,C 180,E1 -15509.651,E2 -15509.651} C_VEL
LIN {X 0,Y 312.514,Z 400.052,A -85,B 0,C 180,E1 -15513.69,E2 -15513.69} C_VEL
LIN {X 0,Y 312.548,Z 400.047,A -85,B 0,C 180,E1 -15517.382,E2 -15517.382} C_VEL
LIN {X 0,Y 312.529,Z 400.037,A -85,B 0,C 180,E1 -15520.703,E2 -15520.703} C_VEL
LIN {X 0,Y 312.53,Z 400.057,A -85,B 0,C 180,E1 -15524.196,E2 -15524.196} C_VEL
LIN {X 0,Y 312.515,Z 400.056,A -85,B 0,C 180,E1 -15527.913,E2 -15527.913} C_VEL
LIN {X 0,Y 312.533,Z 400.057,A -85,B 0,C 180,E1 -15531.911,E2 -15531.911} C_VEL
LIN {X 0,Y 312.532,Z 400.136,A -85,B 0,C 180,E1 -15535.404,E2 -15535.404} C_VEL
LIN {X 0,Y 314.556,Z 408.15,A -85,B 0,C 180,E1 -15538.451,E2 -15538.451} C_VEL
LIN {X 0,Y 316.768,Z 417.944,A -85,B 0,C 180,E1 -15541.872,E2 -15541.872} C_VEL
LIN {X 0,Y 317.23,Z 419.96,A -85,B 0,C 180,E1 -15542.442,E2 -15542.442} C_VEL
LIN {X 0,Y 322.556,Z 432.552,A -85,B 0,C 180,E1 -15543.382,E2 -15543.382} C_VEL
LIN {X 0,Y 326.919,Z 453.306,A -85,B 0,C 180,E1 -15544.364,E2 -15544.364} C_VEL
LIN {X 0,Y 327.968,Z 459.44,A -85,B 0,C 180,E1 -15544.624,E2 -15544.624} C_VEL
LIN {X 0,Y 326.046,Z 527.584,A -85,B 0,C 180,E1 -15546.162,E2 -15546.162} C_VEL
LIN {X 0,Y 325.121,Z 540.714,A -85,B 0,C 180,E1 -15546.682,E2 -15546.682} C_VEL
LIN {X 0,Y 323.803,Z 553.356,A -85,B 0,C 180,E1 -15547.425,E2 -15547.425} C_VEL
LIN {X 0,Y 322.355,Z 565.398,A -85,B 0,C 180,E1 -15548.414,E2 -15548.414} C_VEL
LIN {X 0,Y 320.499,Z 576.87,A -85,B 0,C 180,E1 -15549.629,E2 -15549.629} C_VEL
LIN {X 0,Y 318.7,Z 587.209,A -85,B 0,C 180,E1 -15551.019,E2 -15551.019} C_VEL
LIN {X 0,Y 316.984,Z 596.803,A -85,B 0,C 180,E1 -15552.639,E2 -15552.639} C_VEL
LIN {X 0,Y 315.349,Z 605.546,A -85,B 0,C 180,E1 -15554.489,E2 -15554.489} C_VEL
LIN {X 0,Y 313.746,Z 612.836,A -85,B 0,C 180,E1 -15556.397,E2 -15556.397} C_VEL
LIN {X 0,Y 312.655,Z 618.693,A -85,B 0,C 180,E1 -15558.329,E2 -15558.329} C_VEL
LIN {X 0,Y 311.781,Z 623.328,A -85,B 0,C 180,E1 -15560.267,E2 -15560.267} C_VEL
LIN {X 0,Y 311.193,Z 626.875,A -85,B 0,C 180,E1 -15562.213,E2 -15562.213} C_VEL
LIN {X 0,Y 310.871,Z 629.383,A -85,B 0,C 180,E1 -15564.116,E2 -15564.116} C_VEL
LIN {X 0,Y 310.707,Z 631.07,A -85,B 0,C 180,E1 -15566.109,E2 -15566.109} C_VEL
LIN {X 0,Y 310.656,Z 631.675,A -85,B 0,C 180,E1 -15567.407,E2 -15567.407} C_VEL
LIN {X 0,Y 310.608,Z 631.888,A -85,B 0,C 180,E1 -15568.704,E2 -15568.704} C_VEL
LIN {X 0,Y 310.629,Z 631.671,A -85,B 0,C 180,E1 -15570,E2 -15570} C_VEL
LIN {X 0,Y 310.654,Z 630.072,A -85,B 0,C 180,E1 -15572.594,E2 -15572.594} C_VEL
LIN {X 0,Y 310.688,Z 628.67,A -85,B 0,C 180,E1 -15573.891,E2 -15573.891} C_VEL
LIN {X 0,Y 310.724,Z 626.095,A -85,B 0,C 180,E1 -15575.614,E2 -15575.614} C_VEL
LIN {X 0,Y 311.032,Z 621.714,A -85,B 0,C 180,E1 -15577.792,E2 -15577.792} C_VEL
LIN {X 0,Y 311.623,Z 615.533,A -85,B 0,C 180,E1 -15580.066,E2 -15580.066} C_VEL
